fbRobot.bCNC_4_Reset := 		fbRobot.bCNC_4_Set;

fbRobot.bCNC_5_Reset := 		fbRobot.bCNC_5_Set AND
								stCNC5_Data^.DoorControl_DoorOpened AND
								(NOT stCNC5_Data^.DoorControl_Error) AND 
								stCNC5_Data^.ControlStatus_RobotModeActive
;

fbRobot(
	sName:= 'Fanuc - Satuzó', 
	bEn:= i_bLO2_CNC45, 
	timeBaseState:= T#40S, 
	bAck:= bAckP, 
	bOverride:= nOverride, 
	stEventArray:= arRobotEvents);
END_ACTION

END_PROGRAM

// ---- POUs/FBs/Fanuc/FB_Fanuc.TcPOU
FUNCTION_BLOCK FB_Fanuc
VAR_INPUT
	sName				:STRING;
	bEn					:BOOL;				(* Engedély jel *)
	eCommand			:E_Robot_Command;	(* Végrehajtandó parancsok *)	
	nViseNumber			:BYTE;				(* Satu sorszáma *)	
	nCncNumber			:BYTE;				(* CNC száma; 4 vagy 5 *)
	bVise_1_7_Reset		:BOOL;				(* Handshake *)
	bVise_8_14_Reset	:BOOL;				(* Handshake *)
	bCNC_4_Reset		:BOOL;				(* Handshake *)
	bCNC_5_Reset		:BOOL;				(* Handshake *)
	timeBaseState		:TIME:=T#20S;		(* Alaphelyzet felvételi idő*)
	bAck				:BOOL; 				(* Hibanyugta *)
	bOverride			:BYTE := 10;		(* PLC Override  10 - 100%*)
	stEventArray		:ARRAY [0..nMaxAlarmNr] OF TcEventEntry;	(* Event array definition *)
END_VAR
VAR_OUTPUT
	bReady				:BOOL;				(* Folyamat üzemkész *)
	bBusy				:BOOL;				(* Folyamat aktív *)
	bDone				:BOOL;				(* Folyamat kész *)
	bPendantMode		:BOOL;				(* Teach pendant mód aktív *)
	bVise_1_7_Set		:BOOL;				(* Handshake *)
	bVise_8_14_Set		:BOOL;				(* Handshake *)
	bCNC_4_Set			:BOOL;				(* Handshake *)
	bCNC_5_Set			:BOOL;				(* Handshake *)
	bError				:BOOL;				(* Hiba bit*)
	sError				:STRING(255);		(* Hiba string*)
END_VAR
VAR CONSTANT
	nMaxAlarmNr			:INT := 11;
END_VAR
VAR (* Robot IO *)
	RobotIn				:U_Fanuc_Input;
	RobotOut			:U_Fanuc_Output;
END_VAR
VAR (* State control *)
	tBaseState			:TON;
	tResetFault			:TON;
	tStopCycle			:TON;
	tStartCycle			:TON;
	
	nState				:UDINT;
	sState				:STRING;
	bIsInitalized		:BOOL;
	bRobotReady			:BOOL;
END_VAR
VAR (* Error handling*)
	bErrNotReady		:BOOL;
	bErrBaseTimeout		:BOOL;
	fbAlarmArray		:ARRAY [0..nMaxAlarmNr] OF FB_TcAlarm;
	arrAlarms			:ARRAY [0..nMaxAlarmNr] OF BOOL;
	i					:INT;
	
	//LastStates
	anLastStates				:ARRAY[0..500] OF UDINT;
    iLastStates					:INT;
END_VAR

(*Handshake**************************************************)
bVise_1_7_Set := RobotIn.Status.bVise_1_7_Set;
bVise_8_14_Set := RobotIn.Status.bVise_8_14_Set;
bCNC_4_Set := RobotIn.Status.bCNC_4_Set;
bCNC_5_Set := RobotIn.Status.bCNC_5_Set;
RobotOut.Control.bVise_1_7_Reset := bVise_1_7_Reset;
RobotOut.Control.bVise_8_14_Reset := bVise_8_14_Reset;
RobotOut.Control.bCNC_4_Reset := bCNC_4_Reset;
RobotOut.Control.bCNC_5_Reset := bCNC_5_Reset;

(*Időzítők***************************************************)
tBaseState(IN:= (nState > 0 AND nState < 10000), PT:= timeBaseState);
tResetFault(IN:= RobotOut.Control.bReset, PT:= T#100MS);
tStopCycle(IN:= RobotOut.Control.bCycleStop, PT:= T#100MS);
tStartCycle(IN:= RobotOut.Control.bStart, PT:= T#100MS);

(*Vész rendszer**************************************************)
bRobotReady :=  NOT RobotIn.Status.bControllerEmyStop AND
				NOT RobotIn.Status.bTeachPendantEmyStop AND
				NOT RobotIn.Status.bDeadman AND
				NOT RobotIn.Status.bFence AND
				NOT RobotIn.Status.bEmyStopExternal;
				
(*Hibakezelés************************************************)
IF nState >= 200 AND nState < 150000 AND (RobotIn.Status.bAlarm OR RobotIn.Status.bFault OR NOT bRobotReady) THEN
	bErrNotReady := TRUE;
END_IF

IF tBaseState.Q AND NOT bErrBaseTimeout THEN
	bErrBaseTimeout := TRUE;
END_IF

bError := (RobotIn.Status.bAlarm AND bEn) OR
			RobotIn.Status.bNoPneumatics OR
			RobotIn.Status.bNotCorrectPrg OR
			RobotIn.Status.bNotProductOnRobot OR
			RobotIn.Status.bProductOnRobot OR
			RobotIn.Status.bGripperOpenError OR
			RobotIn.Status.bGripperCloseError OR
			RobotIn.Status.bNotCorrectViseNumber OR
			bErrNotReady OR
			bErrBaseTimeout;

arrAlarms[0] := RobotIn.Status.bNoPneumatics;			
arrAlarms[1] := RobotIn.Status.bNotCorrectPrg;
arrAlarms[2] := RobotIn.Status.bNotProductOnRobot;
arrAlarms[3] := RobotIn.Status.bProductOnRobot;
arrAlarms[4] := RobotIn.Status.bGripperOpenError;
arrAlarms[5] := RobotIn.Status.bGripperCloseError;
arrAlarms[6] := RobotIn.Status.bNotCorrectViseNumber;
arrAlarms[7] := bErrNotReady;
arrAlarms[8] := bErrBaseTimeout;

IF nState > 140 AND nState < 150000 AND bError THEN
	nState := 200000;
END_IF
					
(*State history ************************************************)
IF(nState >= 100) AND (nState <= 20000) THEN
(*Steps before any state*)
	IF anLastStates[0] <> nState THEN
		FOR iLastStates:=500 TO 1 BY -1 DO
			anLastStates[iLastStates]:= anLastStates[iLastStates-1];
		END_FOR
		anLastStates[0]:= nState;
	END_IF
END_IF	

(*Pendant mód ************************************************)
bPendantMode := RobotIn.Status.bPendant;
IF bPendantMode THEN
	nState := 150000;
END_IF

(*Engedélyek *************************************************)
IF (NOT bEn AND NOT bPendantMode) THEN			// nincs ajtókör, és pendantról sem szeretnék használni
	nState := 0;
END_IF

// Enable signals
RobotOut.Control.bZoneEnable := bEn;
RobotOut.Control.bPlcOverride := bOverride;

(*Automata üzem *********************************************)
CASE nState OF
	(* Emergency circuit broken - Base state *)
	0:(* Operation stop - Emergency circuit check *)
		sState := CONCAT(UDINT_TO_STRING(nState) ,' - Vészkör vagy ajtókör bontva - Működtetések törlése');
		RobotOut.Control.bImmediateStop := FALSE;
		RobotOut.Control.bHold := FALSE;
		RobotOut.Control.bSafeSpeed := FALSE;
		RobotOut.Control.bCycleStop := FALSE;
		RobotOut.Control.bReset := FALSE;
		RobotOut.Control.bStart := FALSE;
		RobotOut.Control.bPNS1 := TRUE;
		RobotOut.Control.bPNS2 := FALSE;
		RobotOut.Control.bPNS3 := FALSE;
		RobotOut.Control.bPNS4 := FALSE;
		RobotOut.Control.bPNS5 := FALSE;
		RobotOut.Control.bPNS6 := FALSE;
		RobotOut.Control.bPNS7 := FALSE;
		RobotOut.Control.bPNS8 := FALSE;
		RobotOut.Control.bPnsStrobe := FALSE;
		RobotOut.Control.bEnable := FALSE;
		RobotOut.Control.bHome := FALSE;
		RobotOut.Control.bServiceEnd := FALSE;
		RobotOut.Control.nMode := 0;
		RobotOut.Control.nProgramNumber := 0;
		RobotOut.Control.bProdStart := FALSE;
		RobotOut.Control.bVise_1_7_Reset := FALSE;
		RobotOut.Control.bVise_8_14_Reset := FALSE;
		RobotOut.Control.bCNC_4_Reset := FALSE;
		RobotOut.Control.bCNC_5_Reset := FALSE;
		bErrNotReady := FALSE;
		bErrBaseTimeout := FALSE;
		bReady := FALSE;
		bBusy := FALSE;	
		IF bEn AND bRobotReady THEN
			bBusy := TRUE;
			nState := nState + 20;
		END_IF
		
	20:	
		sState := CONCAT(UDINT_TO_STRING(nState) ,' - Alaphelyzetfelvétel - Robot bekapcsolása');
		RobotOut.Control.bImmediateStop := TRUE;
		RobotOut.Control.bHold := TRUE;
		RobotOut.Control.bSafeSpeed := TRUE;
		RobotOut.Control.bEnable := TRUE;
		IF RobotIn.Status.bFault AND NOT RobotOut.Control.bReset THEN
			RobotOut.Control.bReset := TRUE;	// Ha hiba van -> Reset
		END_IF
		nState := nState + 20;

	40:
		sState := CONCAT(UDINT_TO_STRING(nState) ,' - Alaphelyzet felvétel - Robot hibatörlés');	
		IF tResetFault.Q THEN
			RobotOut.Control.bReset := FALSE;
		END_IF
		IF NOT RobotOut.Control.bReset AND NOT RobotIn.Status.bFault THEN
			nState := nState + 20;
		END_IF

	60:
		sState := CONCAT(UDINT_TO_STRING(nState) ,' - Alaphelyzet felvétel - Várakozás Robot hibatörlésre');	
		IF RobotIn.Status.bCommandEnable AND NOT RobotIn.Status.bFault THEN
			nState := nState + 20;
		END_IF
		
	80:
		sState := CONCAT(UDINT_TO_STRING(nState) ,' - Alaphelyzet felvétel - Robot Cycle Stop');
		RobotOut.Control.bCycleStop := TRUE;
		IF tStopCycle.Q THEN
			RobotOut.Control.bCycleStop := FALSE;
			nState := nState + 20;
		END_IF
	
	100:
		sState := CONCAT(UDINT_TO_STRING(nState) ,' - Alaphelyzet felvétel - Robot Cycle Start');
		RobotOut.Control.bStart := TRUE;
		IF tStartCycle.Q THEN
			RobotOut.Control.bStart := FALSE;
			nState := nState + 20;
		END_IF
		
	120: 
		sState := CONCAT(UDINT_TO_STRING(nState) ,' - Alaphelyzet felvétel - Várakozás Robot Cycle Start-ra');
		IF RobotIn.Status.bBusy AND RobotIn.Status.bProgramEnd THEN
			nState := nState + 20;
		END_IF
		
	140:
		sState := CONCAT(UDINT_TO_STRING(nState) ,' - Alaphelyzet felvétel - Alaphelyzet felvétel - Robot Busy');
		IF RobotIn.Status.bBusy THEN
			RobotOut.Control.bProdStart := TRUE;
			nState := nState + 20;
		END_IF
		
	160:
		sState := CONCAT(UDINT_TO_STRING(nState) ,' - Alaphelyzet felvétel - Robot alaphelyzetbe küldése');	
		RobotOut.Control.nProgramNumber := TO_BYTE(E_Robot_Programs.Home);
		IF RobotOut.Control.nProgramNumber = RobotIn.Status.nProgramNumber THEN
			RobotOut.Control.nProgramNumber := 0;
			nState := nState + 20;
		END_IF
		
	180:
		sState := CONCAT(UDINT_TO_STRING(nState) ,' - Alaphelyzet felvétel - Várakozás a robotprogram végére.');	
		IF RobotIn.Status.bProgramEnd AND NOT RobotIn.Status.bProgramRun THEN
			nState := nState + 20;
		END_IF
		
	200:
		nState := 10000;
		 
(* Alaphelyzet *********************************************************************)
	10000:
		sState := CONCAT(UDINT_TO_STRING(nState) ,' - Alaphelyzet - Várakozás parancsra');
		IF eCommand = E_Robot_Command.NoCommand THEN
			bReady := TRUE;
			bBusy := FALSE;
			bDone := FALSE;
		ELSE
			bReady := TRUE;
			bBusy := TRUE;
			bDone := FALSE;
			IF eCommand = E_Robot_Command.Home THEN			
				nState := 11000;	
			ELSIF eCommand = E_Robot_Command.Wait THEN	
				nState := 12000;
			ELSIF eCommand = E_Robot_Command.Service THEN	
				nState := 13000;
			ELSIF eCommand = E_Robot_Command.Pick_Up_Vise THEN	
				nState := 14000;
			ELSIF eCommand = E_Robot_Command.Put_Down_Vise THEN	
				nState := 15000;
			ELSIF eCommand = E_Robot_Command.Pick_Up_Cnc THEN	
				nState := 16000;
			ELSIF eCommand = E_Robot_Command.Put_Down_Cnc THEN	
				nState := 17000;
			ELSIF eCommand = E_Robot_Command.Move_To_Clean THEN	
				nState := 18000;
			END_IF
		END_IF

{region "Move to Home"} 
	(*-----=== Move to home program végrehajtása ===-----*)
	11000:	
		sState := CONCAT(UDINT_TO_STRING(nState) ,' - Robot alaphelyzetbe küldése');	
			 
		RobotOut.Control.nProgramNumber := TO_BYTE(E_Robot_Programs.Home);
			 
		IF RobotOut.Control.nProgramNumber = RobotIn.Status.nProgramNumber THEN
			RobotOut.Control.nProgramNumber := 0;
			nState := nState + 20;
		END_IF
		
	11020:
		sState := CONCAT(UDINT_TO_STRING(nState) ,' - Várakozás a robotprogram végére.');	
		IF RobotIn.Status.bProgramEnd AND NOT RobotIn.Status.bProgramRun THEN
			nState := nState + 20;
		END_IF
		
	11040:
		sState := CONCAT(UDINT_TO_STRING(nState) ,' - Várakozás mozgásparancs törlésére.');
		bReady := TRUE;
		bBusy := FALSE;
		bDone := TRUE;
		IF eCommand = E_Robot_Command.NoCommand THEN
			nState := 10000;
		END_IF
{enregion}
	 
{region "Move to Wait"}
	(*-----=== Move to wait program végrehajtása ===-----*)
	12000:	
		sState := CONCAT(UDINT_TO_STRING(nState) ,' - Robot várakozó pozícióba küldése');	
				  
		RobotOut.Control.nProgramNumber := TO_BYTE(E_Robot_Programs.Park);
				  
		IF RobotOut.Control.nProgramNumber = RobotIn.Status.nProgramNumber THEN
			RobotOut.Control.nProgramNumber := 0;
			nState := nState + 20;
		END_IF
		
	12020:
		sState := CONCAT(UDINT_TO_STRING(nState) ,' - Várakozás a robotprogram végére.');	
		IF RobotIn.Status.bProgramEnd AND NOT RobotIn.Status.bProgramRun THEN
			nState := nState + 20;
		END_IF
		
	12040:
		sState := CONCAT(UDINT_TO_STRING(nState) ,' - Várakozás mozgásparancs törlésére.');
		bReady := TRUE;
		bBusy := FALSE;
		bDone := TRUE;
		IF eCommand = E_Robot_Command.NoCommand THEN
			nState := 10000;
		END_IF
{enregion}
	 
{region "Move to Service"}
	(*-----=== Move to service program végrehajtása ===-----*)
	13000:	
		sState := CONCAT(UDINT_TO_STRING(nState) ,' - Robot szervíz pozícióba küldése');	
					   
		RobotOut.Control.nProgramNumber := TO_BYTE(E_Robot_Programs.Service);
					   
		IF RobotOut.Control.nProgramNumber = RobotIn.Status.nProgramNumber THEN
			RobotOut.Control.nProgramNumber := 0;
			nState := nState + 20;
		END_IF
		
	13020:
		sState := CONCAT(UDINT_TO_STRING(nState) ,' - Várakozás a robotprogram végére.');	
		IF RobotIn.Status.bProgramEnd AND NOT RobotIn.Status.bProgramRun THEN
			nState := nState + 20;
		END_IF
		
	13040:
		sState := CONCAT(UDINT_TO_STRING(nState) ,' - Várakozás mozgásparancs törlésére.');
		bReady := TRUE;
		bBusy := FALSE;
		bDone := TRUE;
		IF eCommand = E_Robot_Command.NoCommand THEN
			nState := 10000;
		END_IF
{enregion}
	 
{region "Pick up vise"}
	(*-----=== Pick up vise program végrehajtása ===-----*)
	14000:	
		sState := CONCAT(UDINT_TO_STRING(nState) ,' - Felvétel satuzóból');
							
		RobotOut.Control.nViseNumber := nViseNumber;
							
		IF nViseNumber <= 7 THEN
			RobotOut.Control.nProgramNumber := TO_BYTE(E_Robot_Programs.VisePickUp_1_7);
		ELSIF nViseNumber >= 8 THEN
			RobotOut.Control.nProgramNumber := TO_BYTE(E_Robot_Programs.VisePickUp_8_14);
		END_IF
							
		IF RobotOut.Control.nProgramNumber = RobotIn.Status.nProgramNumber THEN
			RobotOut.Control.nProgramNumber := 0;
			nState := nState + 20;
		END_IF
		
	14020:
		sState := CONCAT(UDINT_TO_STRING(nState) ,' - Várakozás a robotprogram végére.');	
		IF RobotIn.Status.bProgramEnd AND NOT RobotIn.Status.bProgramRun THEN
			nState := nState + 20;
		END_IF
		
	14040:
		sState := CONCAT(UDINT_TO_STRING(nState) ,' - Várakozás mozgásparancs törlésére.');
		bReady := TRUE;
		bBusy := FALSE;
		bDone := TRUE;
		IF eCommand = E_Robot_Command.NoCommand THEN
			nState := 10000;
		END_IF
{enregion}
	 
{region "Put down vise"}
	(*-----=== Put down vise program végrehajtása ===-----*)
	15000:	
		sState := CONCAT(UDINT_TO_STRING(nState) ,' - Lerakás satuzóba');
		RobotOut.Control.nViseNumber := nViseNumber;
		IF nViseNumber <= 7 THEN
			RobotOut.Control.nProgramNumber := TO_BYTE(E_Robot_Programs.VisePutDown_1_7);
		ELSIF nViseNumber >= 8 THEN
			RobotOut.Control.nProgramNumber := TO_BYTE(E_Robot_Programs.VisePutDown_8_14);
		END_IF
		IF RobotOut.Control.nProgramNumber = RobotIn.Status.nProgramNumber THEN
			RobotOut.Control.nProgramNumber := 0;
			nState := nState + 20;
		END_IF
		
	15020:
		sState := CONCAT(UDINT_TO_STRING(nState) ,' - Várakozás a robotprogram végére.');	
		IF RobotIn.Status.bProgramEnd AND NOT RobotIn.Status.bProgramRun THEN
			nState := nState + 20;
		END_IF
		
	15040:
		sState := CONCAT(UDINT_TO_STRING(nState) ,' - Várakozás mozgásparancs törlésére.');
		bReady := TRUE;
		bBusy := FALSE;
		bDone := TRUE;
		IF eCommand = E_Robot_Command.NoCommand THEN
			nState := 10000;
		END_IF
{enregion}
	 
{region "Pick up from CNC"}
	(*-----=== Pick up from CNC program végrehajtása ===-----*)
	16000:	
		sState := CONCAT(UDINT_TO_STRING(nState) ,' - Felvétel CNC-ből');
									  
		IF nCncNumber = 4 THEN
			RobotOut.Control.nProgramNumber := TO_BYTE(E_Robot_Programs.VisePickUpFromCnc_4);
		ELSE
			RobotOut.Control.nProgramNumber := TO_BYTE(E_Robot_Programs.VisePickUpFromCnc_5);
		END_IF
									  
		IF RobotOut.Control.nProgramNumber = RobotIn.Status.nProgramNumber THEN
			RobotOut.Control.nProgramNumber := 0;
			nState := nState + 20;
		END_IF
		
	16020:
		sState := CONCAT(UDINT_TO_STRING(nState) ,' - Várakozás a robotprogram végére.');	
		IF RobotIn.Status.bProgramEnd AND NOT RobotIn.Status.bProgramRun THEN
			nState := nState + 20;
		END_IF
		
	16040:
		sState := CONCAT(UDINT_TO_STRING(nState) ,' - Várakozás mozgásparancs törlésére.');
		bReady := TRUE;
		bBusy := FALSE;
		bDone := TRUE;
		IF eCommand = E_Robot_Command.NoCommand THEN
			nState := 10000;
		END_IF
{enregion}
	 
{region "Put down into CNC"}	
	(*-----=== Put down into CNC program végrehajtása ===-----*)
	17000:	
		sState := CONCAT(UDINT_TO_STRING(nState) ,' - Berakás CNC-be');
										   
		IF nCncNumber = 4 THEN
			RobotOut.Control.nProgramNumber := TO_BYTE(E_Robot_Programs.VisePutDownToCnc_4);
		ELSE
			RobotOut.Control.nProgramNumber := TO_BYTE(E_Robot_Programs.VisePutDownToCnc_5);
		END_IF
										   
		IF RobotOut.Control.nProgramNumber = RobotIn.Status.nProgramNumber THEN
			RobotOut.Control.nProgramNumber := 0;
			nState := nState + 20;
		END_IF
		
	17020:
		sState := CONCAT(UDINT_TO_STRING(nState) ,' - Várakozás a robotprogram végére.');	
		IF RobotIn.Status.bProgramEnd AND NOT RobotIn.Status.bProgramRun THEN
			nState := nState + 20;
		END_IF
		
	17040:
		sState := CONCAT(UDINT_TO_STRING(nState) ,' - Várakozás mozgásparancs törlésére.');
		bReady := TRUE;
		bBusy := FALSE;
		bDone := TRUE;
		IF eCommand = E_Robot_Command.NoCommand THEN
			nState := 10000;
		END_IF
{enregion}
	 
{region "Pendant mode"}
(* Pendant mód *********************************************************************)
	150000:	sState := CONCAT(UDINT_TO_STRING(nState) ,' - Pendant mód');
			IF NOT bPendantMode THEN
				RobotOut.Control.bImmediateStop := FALSE;
				RobotOut.Control.bHold := FALSE;
				RobotOut.Control.bZoneEnable := FALSE;
				RobotOut.Control.bEnable := FALSE;
				nState := 0;
			ELSE
				RobotOut.Control.bEnable := TRUE;
				RobotOut.Control.bHold := TRUE;
				RobotOut.Control.bZoneEnable := TRUE;
				RobotOut.Control.bImmediateStop := TRUE;
			END_IF
{endregion}
		
(* Hibakezelés *********************************************************************)
	200000:	sState := CONCAT(UDINT_TO_STRING(nState) ,CONCAT(' - Hiba, ebből az állapotból: ' ,sState));
			bReady := FALSE;
			bBusy := FALSE;	
			nState := nState + 20;

(* Hibakezelés *********************************************************************)
	200020:	
			IF bAck THEN			
				nState := nState + 20;
			END_IF
			
	200040: 
			RobotOut.Control.bImmediateStop := TRUE;
			RobotOut.Control.bReset := TRUE;
			RobotOut.Control.bNotCorrectPrg_Reset := TRUE;
			RobotOut.Control.bNotProductOnRobot_Reset := TRUE;
			RobotOut.Control.bProductOnRobot_Reset := TRUE;
			RobotOut.Control.bGripperOpenError_Reset := TRUE;
			RobotOut.Control.bGripperCloseError_Reset := TRUE;
			RobotOut.Control.bNotCorrectViseNumber_Reset := TRUE;
			nState := nState + 20;
			
	200060:
			IF 	NOT RobotIn.Status.bNoPneumatics AND
				NOT RobotIn.Status.bNotCorrectPrg AND
				NOT RobotIn.Status.bNotProductOnRobot AND
				NOT RobotIn.Status.bProductOnRobot AND
				NOT RobotIn.Status.bGripperOpenError AND
				NOT RobotIn.Status.bGripperCloseError AND
				NOT RobotIn.Status.bNotCorrectViseNumber
			THEN
				nState := nState + 20;
			END_IF	
			
	200080:
			RobotOut.Control.bReset := FALSE;
			RobotOut.Control.bNotCorrectPrg_Reset := FALSE;
			RobotOut.Control.bNotProductOnRobot_Reset := FALSE;
			RobotOut.Control.bProductOnRobot_Reset := FALSE;
			RobotOut.Control.bGripperOpenError_Reset := FALSE;
			RobotOut.Control.bGripperCloseError_Reset := FALSE;
			RobotOut.Control.bNotCorrectViseNumber_Reset := FALSE;
			bErrNotReady := FALSE;
			bErrBaseTimeout := FALSE;
			nState := 0;
ELSE
	sState := CONCAT(UDINT_TO_STRING(nState) ,' - Nem használt állapot');
END_CASE	


(*Hiba string*)
IF bError THEN
	sError := sName;
	FOR i:=0 TO nMaxAlarmNr DO
		IF arrAlarms[i] THEN
			IF (fbAlarmArray[i].eConfirmationState <> 2 AND fbAlarmArray[i].nTimeCleared <> 0 AND fbAlarmArray[i].nTimeConfirmed <> 0) OR //Ha már volt alarm, akkor van bennük érték
				(fbAlarmArray[i].eConfirmationState = 1 AND fbAlarmArray[i].nTimeCleared = 0 AND fbAlarmArray[i].nTimeConfirmed = 0)	//Első futás esetén
			THEN
				fbAlarmArray[i].Raise(0);
			END_IF
		END_IF
	END_FOR 
ELSE
	sError := '';
END_IF

(*Hiba kezelés Tc3_EventLogger*)
IF NOT bIsInitalized THEN
	bIsInitalized := TRUE;
	FOR i:=0 TO nMaxAlarmNr DO
		fbAlarmArray[i].CreateEx(stEventArray[i], TRUE, 0);
	END_FOR
END_IF

(*Hiba törlés (nyugtázott és megszűnt)*)
FOR i:=0 TO nMaxAlarmNr DO
	IF fbAlarmArray[i].eConfirmationState = 3 AND NOT bError THEN
		fbAlarmArray[i].Clear(0, FALSE);
	END_IF
END_FOR

END_FUNCTION_BLOCK

// ---- POUs/Temp/Robot.TcPOU
PROGRAM Robot
VAR
	tResetFault					:TON;
	tStopCycle					:TON;
	tStartCycle					:TON;
END_VAR

(*Bemetek olvasása*******************************************)
stFanucIn := uFanucIn.stFanucIn;
stDigiForceIn := uDigiForceIn.stDigiforce_In;
(*Időzítők***************************************************)
tResetFault(IN:= stFanucOut.stCtrl.bReset, PT:= T#100MS);
tStopCycle(IN:= stFanucOut.stCtrl.bCycleStop, PT:= T#100MS);
tStartCycle(IN:= stFanucOut.stCtrl.bStart, PT:= T#100MS);
(*Triggerek**************************************************)

(*Vész rendszer**********************************************)
bRobotReady := 	NOT stFanucIn.stEmergency.bEMGOP AND
				NOT	stFanucIn.stEmergency.bEMGTP AND
				NOT	stFanucIn.stEmergency.bDEADMAN AND
				NOT	stFanucIn.stEmergency.bFENCE AND
				NOT	stFanucIn.stEmergency.bEMGEX;
				
IF	NOT i_bLOp2 AND
	stRobot.nState > 0 THEN
			stRobot.nState := 0;
END_IF
(*Hibakezelés************************************************)
bRobotAlarm := stRobot.nState > 140 AND	(stFanucIn.stAlarm.bAlarm1 OR
										stFanucIn.stAlarm.bAlarm2 OR
										stFanucIn.stAlarm.bAlarm3 OR
										stFanucIn.stAlarm.bAlarm4 OR
										stFanucIn.stAlarm.bAlarm5 OR
										stFanucIn.stAlarm.bAlarm6);

IF stRobot.nState > 60 AND stRobot.nState < 150000 THEN
	stRobot.nStateLast := stRobot.nState;
	IF	stFanucIn.stCtrl.bFault OR bRobotAlarm OR NOT bRobotReady THEN
			stRobot.nState := 200000;
	END_IF
END_IF
										
(*Engedélyek *************************************************)
IF stRobot.nState <= 10000
	OR stRobot.nState = 150000
	OR stRobot.nState >= 200000
THEN
	stRobot.bManualModeEnable := TRUE;
ELSE
	stRobot.bManualModeEnable := FALSE;
END_IF

IF stRobot.nState = 0
	OR stRobot.nState = 10000
	OR stRobot.nState = 150000
	OR stRobot.nState >= 200000
THEN
	stRobot.bDoorOpenEnable := TRUE;
ELSE
	stRobot.bDoorOpenEnable := FALSE;
END_IF

(*Kézi üzem *************************************************)
IF bManualModeVise and stRobot.nState < 150000 THEN
	stRobot.nState := 150000;
END_IF

(*Automata üzem *********************************************)
CASE stRobot.nState OF
	0:		IF i_bLOp2 AND stProcessReq.bEco THEN			
				stRobot.sState := CONCAT(UDINT_TO_STRING(stRobot.nState) ,' - Robot "ECO" mód aktív - Működtetések törlése');
			ELSE
				stRobot.sState := CONCAT(UDINT_TO_STRING(stRobot.nState) ,' - Vészkör vagy ajtókör bontva - Működtetések törlése');				
			END_IF
			stFanucOut.stCtrl.bImStop := FALSE; 
			stFanucOut.stCtrl.bHold := FALSE; 
			stFanucOut.stCtrl.bSafetyfSpeed := FALSE; 
			stFanucOut.stCtrl.bCycleStop := FALSE; 
			stFanucOut.stCtrl.bReset := FALSE; 
			stFanucOut.stCtrl.bStart := FALSE; 
			stFanucOut.stCtrl.bEnable := FALSE; 
			stFanucOut.stCtrl.bPsr1 := FALSE; 
			stFanucOut.stCtrl.bPsr2 := FALSE; 
			stFanucOut.stCtrl.bPsr3 := FALSE; 
			stFanucOut.stCtrl.bPsr4 := FALSE; 
			stFanucOut.stCtrl.bPsrStrobe := FALSE;
			stFanucOut.stCtrl.bMoveEnable := FALSE; 
			stFanucOut.stCtrl.bServiceEnd := FALSE;
			stFanucOut.stProg.nType := 0;
			stFanucOut.stProg.nMode := 0;
			stFanucOut.stProg.nProgNr := 0;
			stProcessReq.bExecute := FALSE;
			stProcessReq.nProgIdx := 0;
			stRobot.bError := 0;
			IF i_bLOp2 AND bRobotReady AND NOT stProcessReq.bEco THEN
				IF bStepEnable THEN
					stRobot.nState := stRobot.nState + 20;
				END_IF
			END_IF

	20:		stRobot.sState := CONCAT(UDINT_TO_STRING(stRobot.nState) ,' - Alaphelyzet felvétel - Robot bekapcsolása');
			stFanucOut.stCtrl.bImStop := TRUE; 
			stFanucOut.stCtrl.bHold := TRUE; 
			stFanucOut.stCtrl.bSafetyfSpeed := TRUE; 
			stFanucOut.stCtrl.bEnable := TRUE;
			IF stFanucIn.stCtrl.bFault AND NOT stFanucOut.stCtrl.bReset THEN
				stFanucOut.stCtrl.bReset := TRUE;									// Ha hiba van -> Reset
			END_IF
			IF bStepEnable THEN
				stRobot.nState := stRobot.nState + 20;
			END_IF

	40:		stRobot.sState := CONCAT(UDINT_TO_STRING(stRobot.nState) ,' - Alaphelyzet felvétel - Robot hibatörlés');
			IF tResetFault.Q THEN
				stFanucOut.stCtrl.bReset := FALSE;									// Timer-re kell törölni! Hanshake nincs.
			END_IF
			IF NOT stFanucIn.stCtrl.bFault AND NOT stFanucOut.stCtrl.bReset THEN
				IF bStepEnable THEN
					stRobot.nState := stRobot.nState + 20;							// Ha se hiba se reset akkor mehet tovább.
				END_IF
			END_IF
			
	60:		stRobot.sState := CONCAT(UDINT_TO_STRING(stRobot.nState) ,' - Alaphelyzet felvétel - Várakozás Robot hibatörlésre');
			IF stFanucIn.stCtrl.bCmdEnable AND NOT stFanucIn.stCtrl.bFault THEN
				IF bStepEnable THEN
					stRobot.nState := stRobot.nState + 20;
				END_IF
			END_IF

	80:		stRobot.sState := CONCAT(UDINT_TO_STRING(stRobot.nState) ,' - Alaphelyzet felvétel - Robot Cycle Stop');
			stFanucOut.stCtrl.bCycleStop := TRUE;
			IF tStopCycle.Q THEN
				stFanucOut.stCtrl.bCycleStop := FALSE;
				IF bStepEnable THEN
					stRobot.nState := stRobot.nState + 20;
				END_IF
			END_IF
	
	100:	stRobot.sState := CONCAT(UDINT_TO_STRING(stRobot.nState) ,' - Alaphelyzet felvétel - Robot Cycle Start');
			stFanucOut.stCtrl.bStart := TRUE;
			IF tStartCycle.Q THEN
				stFanucOut.stCtrl.bStart := FALSE;
				IF bStepEnable THEN
					stRobot.nState := stRobot.nState + 20;
				END_IF
			END_IF

			
	120:	stRobot.sState := CONCAT(UDINT_TO_STRING(stRobot.nState) ,' - Alaphelyzet felvétel - Várakozás Robot Cycle Start-ra');
			IF stFanucIn.stCtrl.bBusy AND stFanucIn.stCtrl.bProgEnd THEN
				IF bStepEnable THEN
					stRobot.nState := stRobot.nState + 20;
				END_IF
			END_IF
			
	140:	stRobot.sState := CONCAT(UDINT_TO_STRING(stRobot.nState) ,' - Alaphelyzet felvétel - Robot Busy');
			IF stFanucIn.stCtrl.bBusy THEN
				stFanucOut.stCtrl.bMoveEnable := TRUE;								// Robot mozgásengedély
				IF bStepEnable THEN
					stRobot.nState := stRobot.nState + 20;
				END_IF
			END_IF
			
	160:	stRobot.sState := CONCAT(UDINT_TO_STRING(stRobot.nState) ,' - Alaphelyzet felvétel - Robot alaphelyzetbe küldése');
			stFanucOut.stProg.nType := 1;
			stFanucOut.stProg.nMode := 1;
			stFanucOut.stProg.nProgNr := 1;
			IF stFanucOut.stProg.nProgNr = stFanucIn.stProg.nActProg THEN
				stFanucOut.stProg.nProgNr := 0;
				IF bStepEnable THEN
					stRobot.nState := stRobot.nState + 20;
				END_IF
			END_IF

	180:	stRobot.sState := CONCAT(UDINT_TO_STRING(stRobot.nState) ,' - Alaphelyzet felvétel - Várakozás a robotprogram végére.');
			IF	stFanucIn.stProg.nActPoint = 1 AND							// A robot a kiválsztott pontban van
				NOT stFanucIn.stCtrl.bProgRun AND							// A program nem fut
				stFanucIn.stCtrl.bProgEnd THEN								// A program végzett
					IF bStepEnable THEN
						stRobot.nState := stRobot.nState + 20;
					END_IF
			END_IF

	200:
			stRobot.nState := 10000;

	(* Alaphelyzet *********************************************************************)
	10000:	stRobot.sState := CONCAT(UDINT_TO_STRING(stRobot.nState) ,' - Alaphelyzet, parancsra vár');
			IF		stProcessReq.bEco THEN									// Eco mode vagy ajtónyitás
						IF bStepEnable THEN
							stRobot.nState := 20000;
						END_IF
			ELSIF	stProcessReq.bExecute THEN								// Program végrehajtás
						IF stProcessReq.nProgIdx > 0 THEN
							IF bStepEnable THEN
								stRobot.nState := 11000;
							END_IF
						ELSE
							stProcessReq.bExecute := FALSE;
						END_IF
			END_IF

(*-----=== Execute robot program ===-----*)			
	11000:	stRobot.sState := CONCAT(UDINT_TO_STRING(stRobot.nState) ,arrFanucReq[stProcessReq.nProgIdx].sName);
			stFanucOut.stProg.nType := word_to_byte(stP0.stFixtureData.nPcbType);
			stFanucOut.stProg.nMode := 1;
			stFanucOut.stProg.nProgNr := arrFanucReq[stProcessReq.nProgIdx].nProgNr;
			IF (stFanucOut.stProg.nProgNr = stFanucIn.stProg.nActProg) AND											//	A programot tükrözze vissza a robot és	(* Z.Zs. 2022.05.10. *)
			   (stFanucIn.stCtrl.bProgRun AND NOT stFanucIn.stCtrl.bProgEnd) THEN									//	indúljon el a mozgás is, mert a profinet és a PLC elég gyors ahoz, hogy a robotba még ne indúljon el a mozgás!!!!! 
				stProcessReq.nProgIdx := 0;
				IF stProcessReq.nProgIdx2 <> 0 THEN
					stFanucOut.stProg.nProgNr := arrFanucReq[stProcessReq.nProgIdx2].nProgNr;
					IF bStepEnable THEN
						stRobot.nState := stRobot.nState + 20;
					END_IF
				ELSE
					stFanucOut.stProg.nProgNr := 0;
					IF bStepEnable THEN
						stRobot.nState := stRobot.nState + 40;
					END_IF
				END_IF		
			END_IF
			
	11020:	stRobot.sState := CONCAT(UDINT_TO_STRING(stRobot.nState) ,arrFanucReq[stProcessReq.nProgIdx2].sName);
			IF stFanucOut.stProg.nProgNr = stFanucIn.stProg.nActProg THEN
				stProcessReq.nProgIdx2 := 0;
				stFanucOut.stProg.nProgNr := 0;
				IF bStepEnable THEN
					stRobot.nState := stRobot.nState + 20;
				END_IF
			END_IF

	11040:	stRobot.sState := CONCAT(UDINT_TO_STRING(stRobot.nState) ,' - Várakozás a robotprogram végére.');
			IF	NOT stFanucIn.stCtrl.bProgRun AND stFanucIn.stCtrl.bProgEnd THEN
				IF bStepEnable THEN
					stRobot.nState := stRobot.nState + 20;
				END_IF
			END_IF
	
	11060:	
			stRobot.nState := 50000;

(*-----=== ECO mode ===-----*)
	20000:	stRobot.sState := CONCAT(UDINT_TO_STRING(stRobot.nState) ,' - Robot Cycle Stop');
			stFanucOut.stCtrl.bCycleStop := TRUE;
			stFanucOut.stCtrl.bMoveEnable := FALSE;
			IF tStopCycle.Q THEN
				stFanucOut.stCtrl.bCycleStop := FALSE;
				IF bStepEnable THEN
					stRobot.nState := stRobot.nState + 20;
				END_IF
			END_IF

	20020:	stRobot.sState := CONCAT(UDINT_TO_STRING(stRobot.nState) ,' - Robot kikapcsolása');
			stFanucOut.stCtrl.bImStop := FALSE; 
			stFanucOut.stCtrl.bHold := FALSE; 
			stFanucOut.stCtrl.bSafetyfSpeed := FALSE; 
			stFanucOut.stCtrl.bEnable := FALSE;
			IF bStepEnable THEN
				stRobot.nState := 0;
			END_IF			
		
	50000:
			stProcessReq.nProgIdx := 0;
			stProcessReq.bExecute := FALSE;
			stRobot.nState := 10000;
	

	(* Kézi üzem *********************************************************************)
	150000:	stRobot.sState := CONCAT(UDINT_TO_STRING(stRobot.nState) ,' - Kézi üzem');
			IF NOT bManualModeVise THEN
				stRobot.nState := 0;
			ELSIF	stProcessReq.bExecute AND NOT bRobotAlarm AND bRobotReady THEN							// Program végrehajtás
						IF stProcessReq.nProgIdx > 0 THEN
							IF bStepEnable THEN
								stRobot.nState := 151000;
							END_IF
						ELSE
							stProcessReq.bExecute := FALSE;
						END_IF
			ELSIF bRobotAlarm THEN
					stRobot.nState := 152000;
			END_IF

(*-----=== Execute robot program ===-----*)			
	151000:	stRobot.sState := CONCAT(UDINT_TO_STRING(stRobot.nState) ,arrFanucReq[stProcessReq.nProgIdx].sName);
			stFanucOut.stProg.nType := WORD_TO_BYTE(stP0.stFixtureData.nPcbType);
			stFanucOut.stProg.nMode := 1;
			stFanucOut.stProg.nProgNr := arrFanucReq[stProcessReq.nProgIdx].nProgNr;
			IF stFanucOut.stProg.nProgNr = stFanucIn.stProg.nActProg THEN
				stFanucOut.stProg.nProgNr := 0;
				IF bStepEnable THEN
					stRobot.nState := stRobot.nState + 20;
				END_IF
			END_IF

	151020:	stRobot.sState := CONCAT(UDINT_TO_STRING(stRobot.nState) ,' - Várakozás a robotprogram végére.');
			IF	(NOT stFanucIn.stCtrl.bProgRun AND stFanucIn.stCtrl.bProgEnd) OR bRobotAlarm OR NOT bRobotReady THEN
				IF bStepEnable THEN
					stRobot.nState := stRobot.nState + 20;
				END_IF
			END_IF
	
	151040:
			stProcessReq.bExecute := FALSE;
			stRobot.nState := 150000;

(*-----=== Robot alarm törlése ===-----*)
	152000:
			stFanucOut.stAlarm.bAlarm1 := stFanucIn.stAlarm.bAlarm1;
			stFanucOut.stAlarm.bAlarm2 := stFanucIn.stAlarm.bAlarm2;
			stFanucOut.stAlarm.bAlarm3 := stFanucIn.stAlarm.bAlarm3;
			stFanucOut.stAlarm.bAlarm4 := stFanucIn.stAlarm.bAlarm4;
			stFanucOut.stAlarm.bAlarm5 := stFanucIn.stAlarm.bAlarm5;
			stFanucOut.stAlarm.bAlarm6 := stFanucIn.stAlarm.bAlarm6;
			IF NOT bRobotAlarm THEN
				stProcessReq.bExecute := FALSE;
				stRobot.nState := 150000;
			END_IF
	

	(* Hibakezelés *********************************************************************)
	200000:	stRobot.sState := CONCAT(UDINT_TO_STRING(stRobot.nState) ,CONCAT(' - Hiba, ebből az állapotból: ' ,stRobot.sState));
			stRobot.bError := TRUE;
			stRobot.nState := stRobot.nState + 20;

	(* Hibakezelés *********************************************************************)
	200020:	IF bAckP THEN
				stRobot.nState := stRobot.nState + 20;
			END_IF
			

	200040:	stFanucOut.stAlarm.bAlarm1 := stFanucIn.stAlarm.bAlarm1;
			stFanucOut.stAlarm.bAlarm2 := stFanucIn.stAlarm.bAlarm2;
			stFanucOut.stAlarm.bAlarm3 := stFanucIn.stAlarm.bAlarm3;
			stFanucOut.stAlarm.bAlarm4 := stFanucIn.stAlarm.bAlarm4;
			stFanucOut.stAlarm.bAlarm5 := stFanucIn.stAlarm.bAlarm5;
			stFanucOut.stAlarm.bAlarm6 := stFanucIn.stAlarm.bAlarm6;
			IF NOT bRobotAlarm THEN
				stRobot.nState := stRobot.nState + 20;
			END_IF
				
	200060:
				CASE stRobot.nStateLast OF
					(* Alaphelyzet felvétel folyamán *)
					0..9999:	stRobot.nState := 0;
				ELSE 			stRobot.nState := 0;
				END_CASE
				stRobot.bError := FALSE;
ELSE
	stRobot.sState := CONCAT(UDINT_TO_STRING(stRobot.nState) ,' - Nem használt állapot');
END_CASE


(*Robot handshake********************************************)
HandShake();
(*Kimetek írása**********************************************)
uFanucOut.stFanucOut := stFanucOut;
uDigiForceOut.stDigiforce_Out := stDigiForceOut;

ACTION HandShake:
stFanucOut.stHandShake.bFeederEnable := stFanucIn.stHandShake.bFeederReq;
stFanucOut.stHandShake.bPositioner1Enable := stFanucIn.stHandShake.bPositioner1Req;
stFanucOut.stHandShake.bPositioner2Enable := stFanucIn.stHandShake.bPositioner2Req;
stFanucOut.stHandShake.bFixtureAreaEnable := stFanucIn.stHandShake.bFixtureAreaReq;
stFanucOut.stHandShake.bPositioner1Open := stFanucIn.stHandShake.bPositioner1OpenReq AND fbP0Positioner1.bBasePosStab AND fbP0Positioner2.bBasePosStab;
stFanucOut.stHandShake.bPositioner2Open := stFanucIn.stHandShake.bPositioner2OpenReq AND fbP0Positioner3.bBasePosStab AND fbP0Positioner4.bBasePosStab;
END_ACTION

END_PROGRAM

// ---- POUs/Robot7AxisStation/Robot7AxisProgram.TcPOU
PROGRAM Robot7AxisProgram
VAR	(* Control *)
	nState						: UDINT;
	nStatePrevious				: UDINT;
	sState						: STRING(500);
	bError						: BOOL;
	fbCycleTime					: TON;
	nCycleTime					: REAL;
END_VAR
VAR //LastStates
	anLastStates				:ARRAY[0..500] OF UDINT;
    iLastStates					:INT;
END_VAR
VAR (* Robot *)
	fbRobot						: FB_Fanuc_CNC;
	arRobotEvents				: ARRAY [0..15] OF TcEventEntry;
END_VAR
VAR (* Test variables *)
	nOverride					: BYTE := 30;
	bTestEnable					: BOOL;
	nTestIndex					: BYTE;
	nTestCncIndex				: BYTE;
	bCamTest					: BOOL;
	rtCamReset					: R_TRIG;
	nProgNr						: UINT;
	nDimX						: LREAL;
	nDimY						: LREAL;
	nDimZ						: LREAL;
	nPosX						: LREAL;
	nPosY						: LREAL;
	nWeight						: UINT;
	nTorque						: REAL;
	nErrorId					: UDINT;
	ePath						: E_CNC_Robot_Path;
END_VAR
VAR	(*Communication with CNC-s*)
	bStartCNC1					:	BOOL;
	bStartCNC2					:	BOOL;
	bStartCNC3					:	BOOL;
	nPlaceBackFromThisCNC		:	BYTE;
END_VAR
VAR // MySQL
	
END_VAR

MySQL();
Camera();
rtCamReset(CLK:= bCamTest);

IF rtCamReset.Q THEN
		fb3DCam.ResetCam();
END_IF
IF bCamTest THEN
	IF fb3DCam.CamCheck(nProgNr, nDimX, nDimY, nDimZ, nErrorId) THEN
		bCamTest := FALSE;
	END_IF
END_IF

(*Error handling*)
IF nState > 0 AND nState < 150000 THEN
	nStatePrevious := nState;
END_IF

(*Maintance*)
IF bManualMode THEN
	nState := 150000;
END_IF

(*Emergency*)
IF NOT i_bLO1_Main THEN
	nState := 0;
END_IF

(*Last states*)
IF(nState >= 1000) AND (nState < 150000) THEN
(*Steps before any state*)
	IF anLastStates[0] <> nState THEN
		FOR iLastStates:=500 TO 1 BY -1 DO
			anLastStates[iLastStates]:= anLastStates[iLastStates-1];
		END_FOR
		anLastStates[0]:= nState;
	END_IF
END_IF	

IF fbRobot.bError
THEN
	bError  :=  TRUE;
END_IF


(*Yet, constantly write the offset to the used value, because it is the only needed offset now AT 2023.11.17.*)
nPosX := 62.5;
nPosY := (nDimX+4)/2+1;


CASE nState OF
{region "Alaphelyzet felvétel"}
	(****************************************************************************************)
	(******************************* Alaphelyzetfelvétel ************************************)
	(****************************************************************************************)	
	0:		(*-----=== Kimenetek törlése ===-----*)
		sState := CONCAT(UDINT_TO_STRING(nState) ,' - A biztonsági kör nem aktív');
			 
		fbRobot.eCommand := E_CNC_Robot_Command.NoCommand;
		bStartCNC1 := FALSE;
		bStartCNC2 := FALSE;
		bStartCNC3 := FALSE;	
		nPlaceBackFromThisCNC := 0;
			 
		IF i_bLO1_Main AND NOT bManualMode AND NOT fbRobot.bPendantMode THEN
			nState := nState + 20;
		END_IF

	20: 
		sState := CONCAT(UDINT_TO_STRING(nState) ,' - Robot alaphelyzetfelvétel');
		fbRobot.eCommand := E_CNC_Robot_Command.Home;
		IF NOT fbRobot.bBusy AND fbRobot.bReady THEN
			fbRobot.eCommand := E_CNC_Robot_Command.NoCommand;
			nState := nState + 20;
		END_IF

	40:
		nState := 10000;
{endregion}
	 

	10000:
		nState := 10500;
		
	10500:	
		sState := CONCAT(UDINT_TO_STRING(nState) ,' - Paletta kivétel-beküldés ellenőrzés');
		
		//Mi van ha megszakad a folyamat valami maitt?  Akkor is jó ha itt kezd? 
		
		IF stDutData_Cnc1.bDone AND (CNC_1.stCNC_Data^.DoorControl_DoorOpened AND (NOT CNC_1.bCNCHandshakeTimeout)) AND ((fbLift_1A.nTagID = stDutData_Cnc1.nPaletteId)OR(fbLift_1B.nTagID = stDutData_Cnc1.nPaletteId))THEN	//CNC Done, and CNC Door Opened
			
			
			IF fbLift_1A.nTagID = stDutData_Cnc1.nPaletteId THEN	//Decide that what lift should be used
				ePath := E_CNC_Robot_Path.CNC1_to_Lift1A;
				nPlaceBackFromThisCNC := 1;
				nState := 11000;
			ELSIF fbLift_1B.nTagID = stDutData_Cnc1.nPaletteId THEN
				ePath := E_CNC_Robot_Path.CNC1_to_Lift1B;
				nPlaceBackFromThisCNC := 2;
				nState := 11000;
			ELSE
				sState := CONCAT(UDINT_TO_STRING(nState) ,' - Ismeretlen cél lift paletta lerakáskor CNC 1 - Paletta Lift 1 A-B között');
			END_IF
			
		ELSIF stDutData_Cnc2.bDone AND (CNC_2.stCNC_Data^.DoorControl_DoorOpened AND (NOT CNC_2.bCNCHandshakeTimeout)) AND ((fbLift_2A.nTagID = stDutData_Cnc2.nPaletteId)OR(fbLift_2B.nTagID = stDutData_Cnc2.nPaletteId))THEN //CNC Done, and CNC Door Opened
			
			
			IF fbLift_2A.nTagID = stDutData_Cnc2.nPaletteId THEN	//Decide that what lift should be used
				ePath := E_CNC_Robot_Path.CNC2_to_Lift2A;
				nPlaceBackFromThisCNC := 3;
				nState := 11000;
			ELSIF fbLift_2B.nTagID = stDutData_Cnc2.nPaletteId THEN
				ePath := E_CNC_Robot_Path.CNC2_to_Lift2B;
				nPlaceBackFromThisCNC := 4;
				nState := 11000;
			ELSE
				sState := CONCAT(UDINT_TO_STRING(nState) ,' - Ismeretlen cél lift paletta lerakáskor CNC 2 - Paletta Lift 2 A-B között');
			END_IF
		
		ELSIF stDutData_Cnc3.bDone AND (CNC_3.stCNC_Data^.DoorControl_DoorOpened AND (NOT CNC_3.bCNCHandshakeTimeout)) AND ((fbLift_3A.nTagID = stDutData_Cnc3.nPaletteId)OR(fbLift_3B.nTagID = stDutData_Cnc3.nPaletteId))THEN //CNC Done, and CNC Door Opened
				
			nPlaceBackFromThisCNC := 3;
			IF fbLift_3A.nTagID = stDutData_Cnc3.nPaletteId THEN	//Decide that what lift should be used
				ePath := E_CNC_Robot_Path.CNC3_to_Lift3A;
				nPlaceBackFromThisCNC := 5;
				nState := 11000;
			ELSIF fbLift_3B.nTagID = stDutData_Cnc3.nPaletteId THEN
				ePath := E_CNC_Robot_Path.CNC3_to_Lift3B;
				nPlaceBackFromThisCNC := 6;
				nState := 11000;
			ELSE
				sState := CONCAT(UDINT_TO_STRING(nState) ,' - Ismeretlen cél lift paletta lerakáskor CNC 3 - Paletta Lift 3 A-B között');
			END_IF	
			
		
		ELSIF  (NOT CNC_1.bCNCRunning) AND (CNC_1.stCNC_Data^.DoorControl_DoorOpened AND (NOT CNC_1.bCNCHandshakeTimeout)) AND (GVL_Palette.arrPalette[fbLift_1A.nTagID].nState = 3) THEN //Pallet is at the stopper, CNC not running, CNC door is opened
		 		stDutData_Cnc1 := GVL_Palette.arrPalette[fbLift_1A.nTagID];
				ePath := E_CNC_Robot_Path.Lift1A_to_CNC1;
				bStartCNC1 := TRUE;
				nState := 11000;
		ELSIF  (NOT CNC_1.bCNCRunning) AND (CNC_1.stCNC_Data^.DoorControl_DoorOpened AND (NOT CNC_1.bCNCHandshakeTimeout)) AND (GVL_Palette.arrPalette[fbLift_1B.nTagID].nState = 3 ) THEN //Pallet is at the stopper, CNC not running, CNC door is opened
		 		stDutData_Cnc1 := GVL_Palette.arrPalette[fbLift_1B.nTagID];
				ePath := E_CNC_Robot_Path.Lift1B_to_CNC1;
				bStartCNC1 := TRUE;
				nState := 11000;
			
			
		ELSIF  (NOT CNC_2.bCNCRunning) AND (CNC_2.stCNC_Data^.DoorControl_DoorOpened AND (NOT CNC_2.bCNCHandshakeTimeout)) AND (GVL_Palette.arrPalette[fbLift_2A.nTagID].nState = 3)THEN //Pallet is at the stopper, CNC not running, CNC door is opened
		 		stDutData_Cnc2 := GVL_Palette.arrPalette[fbLift_2A.nTagID];
				ePath := E_CNC_Robot_Path.Lift2A_to_CNC2;
				bStartCNC2 := TRUE;
				nState := 11000;
		ELSIF  (NOT CNC_2.bCNCRunning) AND (CNC_2.stCNC_Data^.DoorControl_DoorOpened AND (NOT CNC_2.bCNCHandshakeTimeout)) AND (GVL_Palette.arrPalette[fbLift_2B.nTagID].nState = 3)THEN //Pallet is at the stopper, CNC not running, CNC door is opened
		 		stDutData_Cnc2 := GVL_Palette.arrPalette[fbLift_2B.nTagID];
				ePath := E_CNC_Robot_Path.Lift2B_to_CNC2;
				bStartCNC2 := TRUE;
				nState := 11000;
			
			
		ELSIF  (NOT CNC_3.bCNCRunning) AND (CNC_3.stCNC_Data^.DoorControl_DoorOpened AND (NOT CNC_3.bCNCHandshakeTimeout)) AND (GVL_Palette.arrPalette[fbLift_3A.nTagID].nState = 3) THEN //Pallet is at the stopper, CNC not running, CNC door is opened
		 		stDutData_Cnc3 := GVL_Palette.arrPalette[fbLift_3A.nTagID];
				ePath := E_CNC_Robot_Path.Lift3A_to_CNC3;
				bStartCNC3 := TRUE;
				nState := 11000;
		ELSIF  (NOT CNC_3.bCNCRunning) AND (CNC_3.stCNC_Data^.DoorControl_DoorOpened AND (NOT CNC_3.bCNCHandshakeTimeout)) AND (GVL_Palette.arrPalette[fbLift_3B.nTagID].nState = 3) THEN //Pallet is at the stopper, CNC not running, CNC door is opened
		 		stDutData_Cnc3 := GVL_Palette.arrPalette[fbLift_3B.nTagID];
				ePath := E_CNC_Robot_Path.Lift3B_to_CNC3;
				bStartCNC3 := TRUE;
				nState := 11000;
		END_IF
		

		
{region "Alaphelyzet"}
	(****************************************************************************************)
	(*********************************** Alaphelyzet ****************************************)
	(****************************************************************************************)	
	11000:		(* -----=== Várakozás parancsra ===----- *)
		sState := CONCAT(UDINT_TO_STRING(nState) ,' - Alaphelyzet');
		CASE ePath OF
			E_CNC_Robot_Path.Lift1A_to_CNC1:
												nProgNr := 1;
												fbRobot.nCncNumber := 1;
												fbRobot.eLifterNumber := E_Lifter.Lifter_1A;
												nDimX := stDutData_Cnc1.nDimX;
												nDimY := stDutData_Cnc1.nDimY;
												nDimZ := stDutData_Cnc1.nDimZ;
												nPosX := stDutData_Cnc1.nPosX;
												nPosY := stDutData_Cnc1.nPosY;
												nWeight := stDutData_Cnc1.nWeight;
												nTorque := stDutData_Cnc1.nTorque;
//												stDutData_Cnc1.nDutId := 1;
												nState := 20000;
			E_CNC_Robot_Path.CNC1_to_Lift1A:
												fbRobot.nCncNumber := 1;
												fbRobot.eLifterNumber := E_Lifter.Lifter_1A;
												fbRobot.nOffset_X := nPosX;
												fbRobot.nOffset_Y := nPosY;
												fbRobot.nWeight := stDutData_Cnc1.nWeight;	
												nState := 30000;

			E_CNC_Robot_Path.Lift1B_to_CNC1:
												nProgNr := 2;
												fbRobot.nCncNumber := 1;
												fbRobot.eLifterNumber := E_Lifter.Lifter_1B;
												nDimX := stDutData_Cnc1.nDimX;
												nDimY := stDutData_Cnc1.nDimY;
												nDimZ := stDutData_Cnc1.nDimZ;
												nPosX := stDutData_Cnc1.nPosX;
												nPosY := stDutData_Cnc1.nPosY;
												nWeight := stDutData_Cnc1.nWeight;
												nTorque := stDutData_Cnc1.nTorque;
//												stDutData_Cnc1.nDutId := 1;
												nState := 20000;

			E_CNC_Robot_Path.CNC1_to_Lift1B:
												fbRobot.nCncNumber := 1;
												fbRobot.eLifterNumber := E_Lifter.Lifter_1B;
												fbRobot.nOffset_X := nPosX;
												fbRobot.nOffset_Y := nPosY;
												fbRobot.nWeight := stDutData_Cnc1.nWeight;
												nState := 30000;
													 
														  
															   
																	
																		 
													 
			E_CNC_Robot_Path.Lift2A_to_CNC2:
												nProgNr := 3;
												fbRobot.nCncNumber := 2;
												fbRobot.eLifterNumber := E_Lifter.Lifter_2A;
												nDimX := stDutData_Cnc2.nDimX;
												nDimY := stDutData_Cnc2.nDimY;
												nDimZ := stDutData_Cnc2.nDimZ;
												nPosX := stDutData_Cnc2.nPosX;
												nPosY := stDutData_Cnc2.nPosY;
												nWeight := stDutData_Cnc2.nWeight;
												nTorque := stDutData_Cnc2.nTorque;
//												stDutData_Cnc2.nDutId := 1;
												nState := 20000;
			E_CNC_Robot_Path.CNC2_to_Lift2A:
												fbRobot.nCncNumber := 2;
												fbRobot.eLifterNumber := E_Lifter.Lifter_2A;
												fbRobot.nOffset_X := nPosX;
												fbRobot.nOffset_Y := nPosY;
												fbRobot.nWeight := stDutData_Cnc2.nWeight;	
												nState := 30000;

			E_CNC_Robot_Path.Lift2B_to_CNC2:
												nProgNr := 4;
												fbRobot.nCncNumber := 2;
												fbRobot.eLifterNumber := E_Lifter.Lifter_2B;
												nDimX := stDutData_Cnc2.nDimX;
												nDimY := stDutData_Cnc2.nDimY;
												nDimZ := stDutData_Cnc2.nDimZ;
												nPosX := stDutData_Cnc2.nPosX;
												nPosY := stDutData_Cnc2.nPosY;
												nWeight := stDutData_Cnc2.nWeight;
												nTorque := stDutData_Cnc2.nTorque;
//												stDutData_Cnc2.nDutId := 1;
												nState := 20000;

			E_CNC_Robot_Path.CNC2_to_Lift2B:
												fbRobot.nCncNumber := 2;
												fbRobot.eLifterNumber := E_Lifter.Lifter_2B;
												fbRobot.nOffset_X := nPosX;
												fbRobot.nOffset_Y := nPosY;
												fbRobot.nWeight := stDutData_Cnc2.nWeight;
												nState := 30000;
													 
														  
															   
																	
																		 
																			  
																				   
			E_CNC_Robot_Path.Lift3A_to_CNC3:
												nProgNr := 5;
												fbRobot.nCncNumber := 3;
												fbRobot.eLifterNumber := E_Lifter.Lifter_3A;
												nDimX := stDutData_Cnc3.nDimX;
												nDimY := stDutData_Cnc3.nDimY;
												nDimZ := stDutData_Cnc3.nDimZ;
												nPosX := stDutData_Cnc3.nPosX;
												nPosY := stDutData_Cnc3.nPosY;
												nWeight := stDutData_Cnc3.nWeight;
												nTorque := stDutData_Cnc3.nTorque;
//												stDutData_Cnc3.nDutId := 1;
												nState := 20000;
			E_CNC_Robot_Path.CNC3_to_Lift3A:
												fbRobot.nCncNumber := 3;
												fbRobot.eLifterNumber := E_Lifter.Lifter_3A;
												fbRobot.nOffset_X := nPosX;
												fbRobot.nOffset_Y := nPosY;
												fbRobot.nWeight := stDutData_Cnc3.nWeight;	
												nState := 30000;

			E_CNC_Robot_Path.Lift3B_to_CNC3:
												nProgNr := 6;
												fbRobot.nCncNumber := 3;
												fbRobot.eLifterNumber := E_Lifter.Lifter_3B;
												nDimX := stDutData_Cnc3.nDimX;
												nDimY := stDutData_Cnc3.nDimY;
												nDimZ := stDutData_Cnc3.nDimZ;
												nPosX := stDutData_Cnc3.nPosX;
												nPosY := stDutData_Cnc3.nPosY;
												nWeight := stDutData_Cnc3.nWeight;
												nTorque := stDutData_Cnc3.nTorque;
//												stDutData_Cnc3.nDutId := 1;
												nState := 20000;

			E_CNC_Robot_Path.CNC3_to_Lift3B:
												fbRobot.nCncNumber := 3;
												fbRobot.eLifterNumber := E_Lifter.Lifter_3B;
												fbRobot.nOffset_X := nPosX;
												fbRobot.nOffset_Y := nPosY;
												fbRobot.nWeight := stDutData_Cnc3.nWeight;
												nState := 30000;
		END_CASE
{endregion}

{region "bepakolás a CNC-be"}
	(****************************************************************************************)
	(********************************** Kiemelő -> CNC **************************************)
	(****************************************************************************************)
	20000:		(*-----=== Szkennelési pozícióba ===-----*)
		sState := CONCAT(UDINT_TO_STRING(nState) ,' - Robot kamara pozícióba');
		
		bStartCNC1 := FALSE;
		bStartCNC2 := FALSE;
		bStartCNC3 := FALSE;	 
		
		fbRobot.nOffset_X := 0;
		fbRobot.nOffset_Y := 0;
		fbRobot.nOffset_Z := 0;
		fbRobot.nOffset_W := 0;
		fbRobot.nOffset_P := 0;
		fbRobot.nOffset_R := 0;
		fbRobot.eCommand := E_CNC_Robot_Command.Camera_Lifter;
		IF fbRobot.bBusy THEN
			ePath := E_CNC_Robot_Path.NoPath;
			nState := nState + 20;
		END_IF
		
	20020:		(*-----=== Várakozás Robotmozgásra ===-----*)
		sState := CONCAT(UDINT_TO_STRING(nState) ,' - Várakozáas robot mozgásra');
		IF NOT fbRobot.bBusy THEN
			fbRobot.eCommand := E_CNC_Robot_Command.NoCommand;
			fb3DCam.ResetCam();
			nState := nState + 20;
		END_IF

	20040:		(*-----=== 3D kamera triggerelése ===-----*)
		sState := CONCAT(UDINT_TO_STRING(nState) ,' - 3D kamera triggerelése');
		IF fb3DCam.CamCheck(nProgNr, nDimX, nDimY, nDimZ, nErrorId) THEN
			IF fb3DCam.p_Pass THEN
				nState := nState + 20;
			ELSE
				nState := 200000;
			END_IF
		END_IF

	20060:		(*-----=== Darabfelvétel ===-----*)
		sState := CONCAT(UDINT_TO_STRING(nState) ,' - Robot felvételi pozícióba');
		fbRobot.nOffset_X := fb3DCam.p_PosX;
		fbRobot.nOffset_Y := fb3DCam.p_PosY;
		fbRobot.nOffset_Z := fb3DCam.p_PosZ;
		fbRobot.nOffset_W := fb3DCam.p_PosW;
		fbRobot.nOffset_P := fb3DCam.p_PosP;
		fbRobot.nOffset_R := fb3DCam.p_PosR;
		fbRobot.eCommand := E_CNC_Robot_Command.Pick_Up_Lifter;
		IF fbRobot.bBusy THEN
			nState := nState + 20;
		END_IF
		
	20080:		(*-----=== Várakozás Robotmozgásra ===-----*)
		sState := CONCAT(UDINT_TO_STRING(nState) ,' - Várakozáas robot mozgásra');
		IF NOT fbRobot.bBusy THEN
			fbRobot.eCommand := E_CNC_Robot_Command.NoCommand;
			fb3DCam.ResetCam();
			nState := nState + 20;
		END_IF

	20100:		(*-----=== Darab lerakása ===-----*)
		sState := CONCAT(UDINT_TO_STRING(nState) ,' - Darab lerakása CNC1-be');
		nPosX := 62.5;
		nPosY := (nDimX+4)/2+1;
		fbRobot.nOffset_X := nPosX;
		fbRobot.nOffset_Y := nPosY;
		fbRobot.nOffset_Z := 0;
		fbRobot.nOffset_W := 0;
		fbRobot.nOffset_P := 0;
		fbRobot.nOffset_R := 0;
		fbRobot.eCommand := E_CNC_Robot_Command.Put_Down_CNC;
		IF fbRobot.bBusy THEN
			nState := nState + 20;
		END_IF
		
	20120:		(*-----=== Várakozás Robotmozgásra ===-----*)
		sState := CONCAT(UDINT_TO_STRING(nState) ,' - Várakozáas robot mozgásra');
			   
		IF NOT fbRobot.bBusy THEN
			fbRobot.eCommand := E_CNC_Robot_Command.NoCommand;
			fb3DCam.ResetCam();
			nState := nState + 20;
		END_IF

	20140:		(*-----=== Robot QuickHome pozícióba ===-----*)
		sState := CONCAT(UDINT_TO_STRING(nState) ,' - Robot HOME pozícióba');
		fbRobot.nOffset_X := 0;
		fbRobot.nOffset_Y := 0;
		fbRobot.nOffset_Z := 0;
		fbRobot.nOffset_W := 0;
		fbRobot.nOffset_P := 0;
		fbRobot.nOffset_R := 0;
		fbRobot.eCommand := E_CNC_Robot_Command.QuickHome;
		IF fbRobot.bBusy THEN
			nState := nState + 20;
		END_IF
		
	20160:		(*-----=== Várakozás Robotmozgásra ===-----*)
		sState := CONCAT(UDINT_TO_STRING(nState) ,' - Várakozáas robot mozgásra');
		IF NOT fbRobot.bBusy THEN
			fbRobot.eCommand := E_CNC_Robot_Command.NoCommand;
			fb3DCam.ResetCam();
			nState := nState + 20;
		END_IF

	20180:
		nState := 10000;
{endregion}

{region "kipakolás a CNC-ből"}
	(****************************************************************************************)
	(********************************** CNC -> Kiemelő **************************************)
	(****************************************************************************************)
	30000:		(*-----=== CNC pozícióba ===-----*)
		sState := CONCAT(UDINT_TO_STRING(nState) ,' - Robot CNC pozícióba');
		fbRobot.eCommand := E_CNC_Robot_Command.Pick_Up_CNC;
		IF fbRobot.bBusy THEN
			ePath := E_CNC_Robot_Path.NoPath;
			nState := nState + 20;
		END_IF

	30020:		(*-----=== Várakozás Robotmozgásra ===-----*)
		sState := CONCAT(UDINT_TO_STRING(nState) ,' - Várakozáas robot mozgásra');
		IF NOT fbRobot.bBusy THEN
			fbRobot.eCommand := E_CNC_Robot_Command.NoCommand;
			fb3DCam.ResetCam();
			nState := nState + 20;
		END_IF

	30040:		(*-----=== Lift pozícióba ===-----*)
		sState := CONCAT(UDINT_TO_STRING(nState) ,' - Robot Lift pozícióba');
		fbRobot.eCommand := E_CNC_Robot_Command.Put_Down_Lifter;
		IF fbRobot.bBusy THEN
			nState := nState + 20;
		END_IF

	30060:		(*-----=== Várakozás Robotmozgásra ===-----*)
		sState := CONCAT(UDINT_TO_STRING(nState) ,' - Várakozáas robot mozgásra');
			 
		IF NOT fbRobot.bBusy THEN
					   
			//Liftek visszaküldése alaphelyzetbe			  
			IF nPlaceBackFromThisCNC = 1 THEN
				stDutData_Cnc1.nState.3 := TRUE;
				GVL_Palette.arrPalette[stDutData_Cnc1.nPaletteId].nState.3 := TRUE;
				GVL_Palette.arrPalette[stDutData_Cnc1.nPaletteId].nTarget := 7;
			ELSIF nPlaceBackFromThisCNC = 2 THEN
				stDutData_Cnc1.nState.3 := TRUE;	
				GVL_Palette.arrPalette[stDutData_Cnc1.nPaletteId].nState.3 := TRUE;
				GVL_Palette.arrPalette[stDutData_Cnc1.nPaletteId].nTarget := 7;
					 
			ELSIF nPlaceBackFromThisCNC = 3 THEN
				stDutData_Cnc2.nState.3 := TRUE; 
				GVL_Palette.arrPalette[stDutData_Cnc2.nPaletteId].nState.3 := TRUE;
				GVL_Palette.arrPalette[stDutData_Cnc1.nPaletteId].nTarget := 7;
			ELSIF nPlaceBackFromThisCNC = 4 THEN
				stDutData_Cnc2.nState.3 := TRUE; 
				GVL_Palette.arrPalette[stDutData_Cnc2.nPaletteId].nState.3 := TRUE;
				GVL_Palette.arrPalette[stDutData_Cnc1.nPaletteId].nTarget := 7;
					 
			ELSIF nPlaceBackFromThisCNC = 5 THEN
				stDutData_Cnc3.nState.3 := TRUE; 
				GVL_Palette.arrPalette[stDutData_Cnc3.nPaletteId].nState.3 := TRUE;
				GVL_Palette.arrPalette[stDutData_Cnc1.nPaletteId].nTarget := 7;
			ELSIF nPlaceBackFromThisCNC = 6 THEN
				stDutData_Cnc3.nState.3 := TRUE; 
				GVL_Palette.arrPalette[stDutData_Cnc3.nPaletteId].nState.3 := TRUE;
				GVL_Palette.arrPalette[stDutData_Cnc1.nPaletteId].nTarget := 7;
			END_IF			  
							  		   
		
			fbRobot.eCommand := E_CNC_Robot_Command.NoCommand;
			fb3DCam.ResetCam();
			nState := nState + 20;
		END_IF

	30080:		(*-----=== Robot QuickHome pozícióba ===-----*)
		sState := CONCAT(UDINT_TO_STRING(nState) ,' - Robot HOME pozícióba');
		fbRobot.nOffset_X := 0;
		fbRobot.nOffset_Y := 0;
		fbRobot.nOffset_Z := 0;
		fbRobot.nOffset_W := 0;
		fbRobot.nOffset_P := 0;
		fbRobot.nOffset_R := 0;
		fbRobot.eCommand := E_CNC_Robot_Command.QuickHome;
		IF fbRobot.bBusy THEN
			nState := nState + 20;
		END_IF
		
	30100:		(*-----=== Várakozás Robotmozgásra ===-----*)
		sState := CONCAT(UDINT_TO_STRING(nState) ,' - Várakozáas robot mozgásra');
		IF NOT fbRobot.bBusy THEN
			fbRobot.eCommand := E_CNC_Robot_Command.NoCommand;
			fb3DCam.ResetCam();
			nState := nState + 20;
		END_IF

	30120:
		nState := 10000;


	
	150000: (* Maintenance *)
		sState := CONCAT(UDINT_TO_STRING(nState) ,' - Maintenance');
		IF NOT bManualMode THEN
			nState := 0;
		END_IF
		
	200000:(* Error handling *)
		sState := CONCAT(UDINT_TO_STRING(nState) ,CONCAT(' - Error, from this state: ' , sState));
		nState := 200020;

	200020:(* Error handling *)
		IF bAckP THEN
			CASE nStatePrevious OF
				0..9999: nState := 0;
//				10000..25000: nState := 10000;
//				30000..31000: nState := 30000;
			ELSE nState := 0;
			END_CASE
		END_IF	
		
	ELSE //Not a real step, for test purposes
		sState := CONCAT(UDINT_TO_STRING(nState) ,' - Not a real step, for test purposes');
END_CASE

(*Timers***************************************************)
fbCycleTime(IN:= nState > 10000 AND nState <= 95000, PT:= T#1D, Q=> , ET=> );
IF nState > 10000 AND nState <= 95000 THEN
	nCycleTime := TIME_TO_REAL(fbCycleTime.ET)/1000;
END_IF

Robot();

ACTION Camera:
fb3DCam();
END_ACTION

ACTION MySQL:
;
END_ACTION

ACTION Robot:
arRobotEvents[0] := TC_EVENTS.MyEvents.RobotNoPneumaticsErr;
arRobotEvents[1] := TC_EVENTS.MyEvents.RobotNotCorrectPrgErr;
arRobotEvents[2] := TC_EVENTS.MyEvents.RobotNotProdOnRobotErr;
arRobotEvents[3] := TC_EVENTS.MyEvents.RobotProdOnRobotErr;
arRobotEvents[4] := TC_EVENTS.MyEvents.RobotGripperOpenErr;
arRobotEvents[5] := TC_EVENTS.MyEvents.RobotGripperCloseErr;
arRobotEvents[6] := TC_EVENTS.MyEvents.RobotNotCorrectViseNumberErr;
arRobotEvents[7] := TC_EVENTS.MyEvents.RobotNotReadyErr;
arRobotEvents[8] := TC_EVENTS.MyEvents.RobotBasePosErr;

(*-----=== Gripper jelek kezelése ===-----*)
fbGripperPos1(
	nCalOffset:= 34.9, 
	nReqDistance:= nDimY, 
	bPendantMode:= fbRobot.bPendantMode, 
	bValid=> , 
	nDistance=> , 
	bGripperInPos=> );

fbGripperPos2(
	nCalOffset:= 35, 
	nReqDistance:= nDimY, 
	bPendantMode:= fbRobot.bPendantMode, 
	bValid=> , 
	nDistance=> , 
	bGripperInPos=> );



(*-----=== Hand shake jelek kezelése ===-----*)
fbRobot.bCNC_1_Reset := 			fbRobot.bCNC_1_Set AND				// 05.1	Robot CNC-1-be menne
									i_bRobotDoorOpened_CNC1 AND
									CNC_1.nState = 11100 OR CNC_1.nState = 12000;

fbRobot.bCNC_1_ViseClose_Reset := 	fbRobot.bCNC_1_ViseClose_Set AND	// 05.2	Robot CNC-1 satu zárásra vár
									CNC_1.nState = 11300;

fbRobot.bCNC_1_ViseOpen_Reset := 	fbRobot.bCNC_1_ViseOpen_Set AND		// 05.3	Robot CNC-1 satu nyitásra vár
									CNC_1.nState = 12000;

fbRobot.bCNC_2_Reset := 			fbRobot.bCNC_2_Set AND				// 05.4	Robot CNC-2-be menne
									i_bRobotDoorOpened_CNC2;

fbRobot.bCNC_2_ViseClose_Reset := 	fbRobot.bCNC_2_ViseClose_Set;		// 05.5	Robot CNC-2 satu zárásra vár

fbRobot.bCNC_2_ViseOpen_Reset := 	fbRobot.bCNC_2_ViseOpen_Set;		// 05.6	Robot CNC-2 satu nyitásra vár

fbRobot.bCNC_3_Reset := 			fbRobot.bCNC_3_Set AND				// 05.7	Robot CNC-3-be menne
									i_bRobotDoorOpened_CNC3;

fbRobot.bCNC_3_ViseClose_Reset := 	fbRobot.bCNC_3_ViseClose_Set;		// 05.8	Robot CNC-3 satu zárásra vár
	
fbRobot.bCNC_3_ViseOpen_Reset := 	fbRobot.bCNC_3_ViseOpen_Set;		// 06.1	Robot CNC-3 satu nyitásra vár

fbRobot.bPalette_1_Reset := 		fbRobot.bPalette_1_Set;				// 06.2	Robot Kiemelő 1-hez menne

fbRobot.bPalette_2_Reset := 		fbRobot.bPalette_2_Set;				// 06.3	Robot Kiemelő 2-höz menne

fbRobot.bPalette_3_Reset := 		fbRobot.bPalette_3_Set;				// 06.4	Robot Kiemelő 3-hoz menne

fbRobot.bGripperClosed_Reset := 	fbRobot.bGripperClosed_Set AND		// 06.5	Robot megfogó zárás SET
									(fbGripperPos1.bGripperInPos OR
									fbGripperPos2.bGripperInPos);


fbRobot(
	sName:= 'Fanuc - 7 axis', 
	bEn:= i_bLO2_Main, 
	timeBaseState:= T#40S, 
	bAck:= bAckP, 
	bOverride:= nOverride, 
	stEventArray:= arRobotEvents);
END_ACTION

END_PROGRAM

// ---- POUs/FBs/FanucCNC/FB_Fanuc_CNC.TcPOU
FUNCTION_BLOCK FB_Fanuc_CNC
VAR_INPUT
	sName					:STRING;
	bEn						:BOOL;				(* Engedély jel *)
	eCommand				:E_CNC_Robot_Command;(* Végrehajtandó parancsok *)	
	nCncNumber				:BYTE;				(* CNC gép sorszáma (1-3) *)
	eLifterNumber			:E_Lifter;			(* Kiemelő stípusa *)
	nWeight					:UINT;				(* Offszet érték *)
	nOffset_ID				:UINT;				(* Offszet érték *)
	nOffset_X				:REAL;				(* X tengelyű offszet érték *)
	nOffset_Y				:REAL;				(* Y tengelyű offszet érték *)
	nOffset_Z				:REAL;				(* Z tengelyű offszet érték *)
	nOffset_W				:REAL;				(* W tengelyű offszet érték *)
	nOffset_P				:REAL;				(* P tengelyű offszet érték *)
	nOffset_R				:REAL;				(* R tengelyű offszet érték *)
	bCNC_1_Reset			:BOOL;				(* Handshake *)
	bCNC_1_ViseClose_Reset	:BOOL;				(* Handshake *)
	bCNC_1_ViseOpen_Reset	:BOOL;				(* Handshake *)
	bCNC_2_Reset			:BOOL;				(* Handshake *)
	bCNC_2_ViseClose_Reset	:BOOL;				(* Handshake *)
	bCNC_2_ViseOpen_Reset	:BOOL;				(* Handshake *)
	bCNC_3_Reset			:BOOL;				(* Handshake *)
	bCNC_3_ViseClose_Reset	:BOOL;				(* Handshake *)
	bCNC_3_ViseOpen_Reset	:BOOL;				(* Handshake *)
	bPalette_1_Reset		:BOOL;				(* Handshake *)
	bPalette_2_Reset		:BOOL;				(* Handshake *)
	bPalette_3_Reset		:BOOL;				(* Handshake *)
	bGripperClosed_Reset	:BOOL;				(* Handshake *)
	timeBaseState			:TIME:=T#20S;		(* Alaphelyzet felvételi idő*)
	bAck					:BOOL; 				(* Hibanyugta *)
	bOverride				:BYTE := 10;		(* PLC Override  10 - 100%*)
	stEventArray			:ARRAY [0..nMaxAlarmNr] OF TcEventEntry;	(* Event array definition *)
END_VAR
VAR_OUTPUT
	bReady					:BOOL;				(* Folyamat üzemkész *)
	bBusy					:BOOL;				(* Folyamat aktív *)
	bDone					:BOOL;				(* Folyamat kész *)
	bPendantMode			:BOOL;				(* Teach pendant mód aktív *)
	bCNC_1_Set				:BOOL;				(* Handshake *)
	bCNC_1_ViseClose_Set	:BOOL;				(* Handshake *)
	bCNC_1_ViseOpen_Set		:BOOL;				(* Handshake *)
	bCNC_2_Set				:BOOL;				(* Handshake *)
	bCNC_2_ViseClose_Set	:BOOL;				(* Handshake *)
	bCNC_2_ViseOpen_Set		:BOOL;				(* Handshake *)
	bCNC_3_Set				:BOOL;				(* Handshake *)
	bCNC_3_ViseClose_Set	:BOOL;				(* Handshake *)
	bCNC_3_ViseOpen_Set		:BOOL;				(* Handshake *)
	bPalette_1_Set			:BOOL;				(* Handshake *)
	bPalette_2_Set			:BOOL;				(* Handshake *)
	bPalette_3_Set			:BOOL;				(* Handshake *)
	bGripperClosed_Set		:BOOL;				(* Handshake *)
	bError					:BOOL;				(* Hiba bit*)
	sError					:STRING(255);		(* Hiba string*)
	bZoneCnc1				:BOOL;				(* Robot bent a területen Zone 1*)
	bZoneCnc2				:BOOL;				(* Robot bent a területen Zone 2*)
	bZoneCnc3				:BOOL;				(* Robot bent a területen Zone 3*)
	bZoneLift1				:BOOL;				(* Robot bent a területen Zone 4*)
	bZoneLift2				:BOOL;				(* Robot bent a területen Zone 5*)
	bZoneLift3				:BOOL;				(* Robot bent a területen Zone 6*)
	bZoneGudel				:BOOL;				(* Robot bent a területen Zone 7*)
	bZoneMaster				:BOOL;				(* Robot bent a területen Zone 8*)
	nOffset_ID_Echo			:UINT;				(* Offszet érték *)
	nOffset_X_Echo			:REAL;				(* X tengelyű offszet érték *)
	nOffset_Y_Echo			:REAL;				(* Y tengelyű offszet érték *)
	nOffset_Z_Echo			:REAL;				(* Z tengelyű offszet érték *)
	nOffset_W_Echo			:REAL;				(* W tengelyű offszet érték *)
	nOffset_P_Echo			:REAL;				(* P tengelyű offszet érték *)
	nOffset_R_Echo			:REAL;				(* R tengelyű offszet érték *)
END_VAR
VAR CONSTANT
	nMaxAlarmNr			:INT := 15;
	nDecimalPlaces		:USINT := 3;
END_VAR
VAR (* Robot IO *)
	RobotIn				:U_CNC_Fanuc_Input;
	RobotOut			:U_CNC_Fanuc_Output;
END_VAR
VAR (* State control *)
	tBaseState			:TON;
	tResetFault			:TON;
	tStopCycle			:TON;
	tStartCycle			:TON;
	
	nState				:UDINT;
	sState				:STRING;
	bIsInitalized		:BOOL;
	bRobotReady			:BOOL;
END_VAR
VAR (* Error handling*)
	bErrNotReady		:BOOL;
	bErrBaseTimeout		:BOOL;
	fbAlarmArray		:ARRAY [0..nMaxAlarmNr] OF FB_TcAlarm;
	arrAlarms			:ARRAY [0..nMaxAlarmNr] OF BOOL;
	i					:INT;
	
	//LastStates
	anLastStates				:ARRAY[0..500] OF UDINT;
    iLastStates					:INT;
END_VAR
VAR
// TEST !!!!!!!!!!!!!!!!!!!!!!
	bTestConvert		: BOOL;
END_VAR

(*Test*) //TÖRÖLNI HA MÁR HOMÁR!!!!!!!!!!!!!!!!!!!!!!!!!!!!!!!!!!!!!!!!!!!!!!!!!!!!!!!!!!!!!!!!!!!!!!!!!!!!!!!!!!!!!!!
IF bTestConvert THEN
		REAL_TO_WHOLE_AND_FRACTION(nReal := nOffset_X,
									nWhole => RobotOut.Control.nOffset_X_Whole,
									nFraction => RobotOut.Control.nOffset_X_Fractional);
		REAL_TO_WHOLE_AND_FRACTION(nReal := nOffset_Y,
									nWhole => RobotOut.Control.nOffset_Y_Whole,
									nFraction => RobotOut.Control.nOffset_Y_Fractional);
		REAL_TO_WHOLE_AND_FRACTION(nReal := nOffset_Z,
									nWhole => RobotOut.Control.nOffset_Z_Whole,
									nFraction => RobotOut.Control.nOffset_Z_Fractional);
		REAL_TO_WHOLE_AND_FRACTION(nReal := nOffset_W,
									nWhole => RobotOut.Control.nOffset_W_Whole,
									nFraction => RobotOut.Control.nOffset_W_Fractional);
		REAL_TO_WHOLE_AND_FRACTION(nReal := nOffset_P,
									nWhole => RobotOut.Control.nOffset_P_Whole,
									nFraction => RobotOut.Control.nOffset_P_Fractional);
		REAL_TO_WHOLE_AND_FRACTION(nReal := nOffset_R,
									nWhole => RobotOut.Control.nOffset_R_Whole,
									nFraction => RobotOut.Control.nOffset_R_Fractional);
		bTestConvert := FALSE;
END_IF
(*Offset Echo************************************************)
nOffset_ID_Echo := RobotIn.Status.nOffset_ID;
WHOLE_AND_FRACTION_TO_REAL(nWhole:= RobotIn.Status.nOffset_X_Whole, nFraction:=RobotIn.Status.nOffset_X_Fractional, nReal=> nOffset_X_Echo);
WHOLE_AND_FRACTION_TO_REAL(nWhole:= RobotIn.Status.nOffset_Y_Whole, nFraction:=RobotIn.Status.nOffset_Y_Fractional, nReal=> nOffset_Y_Echo);
WHOLE_AND_FRACTION_TO_REAL(nWhole:= RobotIn.Status.nOffset_Z_Whole, nFraction:=RobotIn.Status.nOffset_Z_Fractional, nReal=> nOffset_Z_Echo);
WHOLE_AND_FRACTION_TO_REAL(nWhole:= RobotIn.Status.nOffset_W_Whole, nFraction:=RobotIn.Status.nOffset_W_Fractional, nReal=> nOffset_W_Echo);
WHOLE_AND_FRACTION_TO_REAL(nWhole:= RobotIn.Status.nOffset_P_Whole, nFraction:=RobotIn.Status.nOffset_P_Fractional, nReal=> nOffset_P_Echo);
WHOLE_AND_FRACTION_TO_REAL(nWhole:= RobotIn.Status.nOffset_R_Whole, nFraction:=RobotIn.Status.nOffset_R_Fractional, nReal=> nOffset_R_Echo);

(*Handshake**************************************************)
bCNC_1_Set := RobotIn.Status.bCNC_1_Set;
bCNC_1_ViseClose_Set := RobotIn.Status.bCNC_1_ViseClose_Set;
bCNC_1_ViseOpen_Set := RobotIn.Status.bCNC_1_ViseOpen_Set;
bCNC_2_Set := RobotIn.Status.bCNC_2_Set;
bCNC_2_ViseClose_Set := RobotIn.Status.bCNC_2_ViseClose_Set;
bCNC_2_ViseOpen_Set := 	RobotIn.Status.bCNC_2_ViseOpen_Set;
bCNC_3_Set := RobotIn.Status.bCNC_3_Set;
bCNC_3_ViseClose_Set := RobotIn.Status.bCNC_3_ViseClose_Set;
bCNC_3_ViseOpen_Set := RobotIn.Status.bCNC_3_ViseOpen_Set;
bPalette_1_Set := RobotIn.Status.bPalette_1_Set;
bPalette_2_Set := RobotIn.Status.bPalette_2_Set;
bPalette_3_Set := RobotIn.Status.bPalette_3_Set;
bGripperClosed_Set := RobotIn.Status.bGripperClosed_Set;
RobotOut.Control.bCNC_1_Reset := bCNC_1_Reset;
RobotOut.Control.bCNC_1_ViseClose_Reset := bCNC_1_ViseClose_Reset;
RobotOut.Control.bCNC_1_ViseOpen_Reset := bCNC_1_ViseOpen_Reset;
RobotOut.Control.bCNC_2_Reset := bCNC_2_Reset;
RobotOut.Control.bCNC_2_ViseClose_Reset := bCNC_2_ViseClose_Reset;
RobotOut.Control.bCNC_2_ViseOpen_Reset := 	bCNC_2_ViseOpen_Reset;
RobotOut.Control.bCNC_3_Reset := bCNC_3_Reset;
RobotOut.Control.bCNC_3_ViseClose_Reset := bCNC_3_ViseClose_Reset;
RobotOut.Control.bCNC_3_ViseOpen_Reset := bCNC_3_ViseOpen_Reset;
RobotOut.Control.bPalette_1_Reset := bPalette_1_Reset;
RobotOut.Control.bPalette_2_Reset := bPalette_2_Reset;
RobotOut.Control.bPalette_3_Reset := bPalette_3_Reset;
RobotOut.Control.bGripperClosed_Reset := bGripperClosed_Reset;
RobotOut.Control.nWeight := nWeight;

(*Zónák******************************************************)
bZoneCnc1 :=  RobotIn.Status.bZone_1_CNC_1;
bZoneCnc2 := RobotIn.Status.bZone_2_CNC_2;
bZoneCnc3 := RobotIn.Status.bZone_3_CNC_3;
bZoneLift1 := RobotIn.Status.bZone_4_Lifter_1;
bZoneLift2 := RobotIn.Status.bZone_5_Lifter_2;
bZoneLift3 := RobotIn.Status.bZone_6_Lifter_3;
bZoneGudel := RobotIn.Status.bZone_7_Gudel;
bZoneMaster := RobotIn.Status.bZone_8_Master;


(*Időzítők***************************************************)
tBaseState(IN:= (nState > 0 AND nState < 10000), PT:= timeBaseState);
tResetFault(IN:= RobotOut.Control.bReset, PT:= T#100MS);
tStopCycle(IN:= RobotOut.Control.bCycleStop, PT:= T#100MS);
tStartCycle(IN:= RobotOut.Control.bStart, PT:= T#100MS);

(*Vész rendszer**************************************************)
bRobotReady :=  NOT RobotIn.Status.bControllerEmyStop AND
				NOT RobotIn.Status.bTeachPendantEmyStop AND
				NOT RobotIn.Status.bDeadman AND
				NOT RobotIn.Status.bFence AND
				NOT RobotIn.Status.bEmyStopExternal;
				
(*Hibakezelés************************************************)
IF nState >= 200 AND nState < 150000 AND (RobotIn.Status.bAlarm OR RobotIn.Status.bFault OR NOT bRobotReady) THEN
	bErrNotReady := TRUE;
ELSIF nState = 40 AND bErrBaseTimeout THEN
	nState := 200000;
END_IF

IF tBaseState.Q AND NOT bErrBaseTimeout THEN
	bErrBaseTimeout := TRUE;
END_IF

bError := (RobotIn.Status.bAlarm AND bEn) OR
			RobotIn.Status.bNoPneumatics OR
			RobotIn.Status.bNotCorrectPrg OR
			RobotIn.Status.bNotProductOnRobot OR
			RobotIn.Status.bProductOnRobot OR
			RobotIn.Status.bGripperOpenError OR
			RobotIn.Status.bGripperCloseError OR
			RobotIn.Status.bOffsetError OR
			RobotIn.Status.bWeightError OR
			bErrNotReady OR
			bErrBaseTimeout;

arrAlarms[0] := RobotIn.Status.bNoPneumatics;			
arrAlarms[1] := RobotIn.Status.bNotCorrectPrg;
arrAlarms[2] := RobotIn.Status.bNotProductOnRobot;
arrAlarms[3] := RobotIn.Status.bProductOnRobot;
arrAlarms[4] := RobotIn.Status.bGripperOpenError;
arrAlarms[5] := RobotIn.Status.bGripperCloseError;
arrAlarms[6] := RobotIn.Status.bOffsetError;
arrAlarms[7] := RobotIn.Status.bWeightError;
arrAlarms[8] := bErrNotReady;
arrAlarms[9] := bErrBaseTimeout;

IF nState > 140 AND nState < 150000 AND bError THEN
	nState := 200000;
END_IF
					
(*State history ************************************************)
IF(nState >= 100) AND (nState <= 20000) THEN
(*Steps before any state*)
	IF anLastStates[0] <> nState THEN
		FOR iLastStates:=500 TO 1 BY -1 DO
			anLastStates[iLastStates]:= anLastStates[iLastStates-1];
		END_FOR
		anLastStates[0]:= nState;
	END_IF
END_IF	

(*Pendant mód ************************************************)
bPendantMode := RobotIn.Status.bPendant;
IF bPendantMode THEN
	nState := 150000;
END_IF

(*Engedélyek *************************************************)
IF (NOT bEn AND NOT bPendantMode) THEN			// nincs ajtókör, és pendantról sem szeretnék használni
	nState := 0;
END_IF

// Enable signals
RobotOut.Control.bZoneEnable := bEn;
RobotOut.Control.bPlcOverride := bOverride;

(*Automata üzem *********************************************)
CASE nState OF
	(* Emergency circuit broken - Base state *)
	0:(* Operation stop - Emergency circuit check *)
		sState := CONCAT(UDINT_TO_STRING(nState) ,' - Vészkör vagy ajtókör bontva - Működtetések törlése');
		RobotOut.Control.bImmediateStop := FALSE;
		RobotOut.Control.bHold := FALSE;
		RobotOut.Control.bSafeSpeed := FALSE;
		RobotOut.Control.bCycleStop := FALSE;
		RobotOut.Control.bReset := FALSE;
		RobotOut.Control.bStart := FALSE;
		RobotOut.Control.bPNS1 := TRUE;
		RobotOut.Control.bPNS2 := FALSE;
		RobotOut.Control.bPNS3 := FALSE;
		RobotOut.Control.bPNS4 := FALSE;
		RobotOut.Control.bPNS5 := FALSE;
		RobotOut.Control.bPNS6 := FALSE;
		RobotOut.Control.bPNS7 := FALSE;
		RobotOut.Control.bPNS8 := FALSE;
		RobotOut.Control.bPnsStrobe := FALSE;
		RobotOut.Control.bEnable := FALSE;
		RobotOut.Control.bHome := FALSE;
		RobotOut.Control.bServiceEnd := FALSE;
		RobotOut.Control.nMode := 0;
		RobotOut.Control.nProgramNumber := 0;
		RobotOut.Control.bProdStart := FALSE;
		RobotOut.Control.bCNC_1_Reset := FALSE;
		RobotOut.Control.bCNC_1_ViseClose_Reset := FALSE;
		RobotOut.Control.bCNC_1_ViseOpen_Reset := FALSE;
		RobotOut.Control.bCNC_2_Reset := FALSE;
		RobotOut.Control.bCNC_2_ViseClose_Reset := FALSE;
		RobotOut.Control.bCNC_2_ViseOpen_Reset := FALSE;
		RobotOut.Control.bCNC_3_Reset := FALSE;
		RobotOut.Control.bCNC_3_ViseClose_Reset := FALSE;
		RobotOut.Control.bCNC_3_ViseOpen_Reset := FALSE;
		RobotOut.Control.bPalette_1_Reset := FALSE;
		RobotOut.Control.bPalette_2_Reset := FALSE;
		RobotOut.Control.bPalette_3_Reset := FALSE;
		RobotOut.Control.bGripperClosed_Reset := FALSE;
		bErrNotReady := FALSE;
		bErrBaseTimeout := FALSE;
		bReady := FALSE;
		bBusy := FALSE;	
		IF bEn AND bRobotReady THEN
			bBusy := TRUE;
			nState := nState + 20;
		END_IF
		
	20:	
		sState := CONCAT(UDINT_TO_STRING(nState) ,' - Alaphelyzetfelvétel - Robot bekapcsolása');
		RobotOut.Control.bImmediateStop := TRUE;
		RobotOut.Control.bHold := TRUE;
		RobotOut.Control.bSafeSpeed := TRUE;
		RobotOut.Control.bEnable := TRUE;
		IF RobotIn.Status.bFault AND NOT RobotOut.Control.bReset THEN
			RobotOut.Control.bReset := TRUE;	// Ha hiba van -> Reset
		END_IF
		nState := nState + 20;

	40:
		sState := CONCAT(UDINT_TO_STRING(nState) ,' - Alaphelyzet felvétel - Robot hibatörlés');	
		IF tResetFault.Q THEN
			RobotOut.Control.bReset := FALSE;
		END_IF
		IF NOT RobotOut.Control.bReset AND NOT RobotIn.Status.bFault THEN
			nState := nState + 20;
		END_IF

	60:
		sState := CONCAT(UDINT_TO_STRING(nState) ,' - Alaphelyzet felvétel - Várakozás Robot hibatörlésre');	
		IF RobotIn.Status.bCommandEnable AND NOT RobotIn.Status.bFault THEN
			nState := nState + 20;
		END_IF
		
	80:
		sState := CONCAT(UDINT_TO_STRING(nState) ,' - Alaphelyzet felvétel - Robot Cycle Stop');
		RobotOut.Control.bCycleStop := TRUE;
		IF tStopCycle.Q THEN
			RobotOut.Control.bCycleStop := FALSE;
			nState := nState + 20;
		END_IF
	
	100:
		sState := CONCAT(UDINT_TO_STRING(nState) ,' - Alaphelyzet felvétel - Robot Cycle Start');
		RobotOut.Control.bStart := TRUE;
		IF tStartCycle.Q THEN
			RobotOut.Control.bStart := FALSE;
			nState := nState + 20;
		END_IF
		
	120: 
		sState := CONCAT(UDINT_TO_STRING(nState) ,' - Alaphelyzet felvétel - Várakozás Robot Cycle Start-ra');
		IF RobotIn.Status.bBusy AND RobotIn.Status.bProgramEnd THEN
			nState := nState + 20;
		END_IF
		
	140:
		sState := CONCAT(UDINT_TO_STRING(nState) ,' - Alaphelyzet felvétel - Alaphelyzet felvétel - Robot Busy');
		IF RobotIn.Status.bBusy THEN
			RobotOut.Control.bProdStart := TRUE;
			nState := nState + 20;
		END_IF
		
	160:
		sState := CONCAT(UDINT_TO_STRING(nState) ,' - Alaphelyzet felvétel - Robot alaphelyzetbe küldése');	
		RobotOut.Control.nProgramNumber := TO_BYTE(E_CNC_Robot_Programs.Home);
		IF RobotOut.Control.nProgramNumber = RobotIn.Status.nProgramNumber THEN
			RobotOut.Control.nProgramNumber := 0;
			nState := nState + 20;
		END_IF
		
	180:
		sState := CONCAT(UDINT_TO_STRING(nState) ,' - Alaphelyzet felvétel - Várakozás a robotprogram végére.');	
		IF RobotIn.Status.bProgramEnd AND NOT RobotIn.Status.bProgramRun THEN
			nState := nState + 20;
		END_IF
		
	200:
		nState := 10000;
		 
(* Alaphelyzet *********************************************************************)
	10000:
		sState := CONCAT(UDINT_TO_STRING(nState) ,' - Alaphelyzet - Várakozás parancsra');
		IF eCommand = E_CNC_Robot_Command.NoCommand THEN
			bReady := TRUE;
			bBusy := FALSE;
			bDone := FALSE;
		ELSE
			bReady := TRUE;
			bBusy := TRUE;
			bDone := FALSE;
			IF eCommand = E_CNC_Robot_Command.Home THEN			
				nState := 11000;	
			ELSIF eCommand = E_CNC_Robot_Command.QuickHome THEN	
				nState := 11500;
			ELSIF eCommand = E_CNC_Robot_Command.Wait THEN	
				nState := 12000;
			ELSIF eCommand = E_CNC_Robot_Command.Service THEN	
				nState := 13000;
			ELSIF eCommand = E_CNC_Robot_Command.Pick_Up_CNC THEN	
				nState := 14000;
			ELSIF eCommand = E_CNC_Robot_Command.Put_Down_CNC THEN	
				nState := 15000;
			ELSIF eCommand = E_CNC_Robot_Command.Pick_Up_Lifter THEN	
				nState := 16000;
			ELSIF eCommand = E_CNC_Robot_Command.Put_Down_Lifter THEN	
				nState := 17000;
			ELSIF eCommand = E_CNC_Robot_Command.Camera_Lifter THEN	
				nState := 18000;
			ELSIF eCommand = E_CNC_Robot_Command.Pick_Up_Master THEN	
				nState := 19000;
			ELSIF eCommand = E_CNC_Robot_Command.Put_Down_Master THEN	
				nState := 20000;
			ELSIF eCommand = E_CNC_Robot_Command.Pick_Up_Master_From_Lifter THEN	
				nState := 21000;
			ELSIF eCommand = E_CNC_Robot_Command.Put_Down_Master_To_Lifter THEN	
				nState := 22000;
			END_IF
		END_IF

{region "Move to Home"} 
	(*-----=== Move to home program végrehajtása ===-----*)
	11000:	
		sState := CONCAT(UDINT_TO_STRING(nState) ,' - Robot alaphelyzetbe küldése');	
		RobotOut.Control.nProgramNumber := TO_BYTE(E_CNC_Robot_Programs.Home);
		IF RobotOut.Control.nProgramNumber = RobotIn.Status.nProgramNumber THEN
			RobotOut.Control.nProgramNumber := 0;
			nState := nState + 20;
		END_IF
		
	11020:
		sState := CONCAT(UDINT_TO_STRING(nState) ,' - Várakozás a robotprogram végére.');	
		IF RobotIn.Status.bProgramEnd AND NOT RobotIn.Status.bProgramRun THEN
			nState := nState + 20;
		END_IF
		
	11040:
		sState := CONCAT(UDINT_TO_STRING(nState) ,' - Várakozás mozgásparancs törlésére.');
		bReady := TRUE;
		bBusy := FALSE;
		bDone := TRUE;
		IF eCommand = E_CNC_Robot_Command.NoCommand THEN
			nState := 10000;
		END_IF
{endregion}

{region "Move to Quick Home"}
	 	(*-----=== Move to quick home program végrehajtása ===-----*)
	11500:	
		sState := CONCAT(UDINT_TO_STRING(nState) ,' - Robot alaphelyzetbe küldése');	
		RobotOut.Control.nProgramNumber := TO_BYTE(E_CNC_Robot_Programs.QuickHome);
		IF RobotOut.Control.nProgramNumber = RobotIn.Status.nProgramNumber THEN
			RobotOut.Control.nProgramNumber := 0;
			nState := nState + 20;
		END_IF
		
	11520:
		sState := CONCAT(UDINT_TO_STRING(nState) ,' - Várakozás a robotprogram végére.');	
		IF RobotIn.Status.bProgramEnd AND NOT RobotIn.Status.bProgramRun THEN
			nState := nState + 20;
		END_IF
		
	11540:
		sState := CONCAT(UDINT_TO_STRING(nState) ,' - Várakozás mozgásparancs törlésére.');
		bReady := TRUE;
		bBusy := FALSE;
		bDone := TRUE;
		IF eCommand = E_CNC_Robot_Command.NoCommand THEN
			nState := 10000;
		END_IF
{endregion}

{region "Move to Wait"}
	(*-----=== Move to wait program végrehajtása ===-----*)
	12000:	
		sState := CONCAT(UDINT_TO_STRING(nState) ,' - Robot várakozó pozícióba küldése');	
		RobotOut.Control.nProgramNumber := TO_BYTE(E_CNC_Robot_Programs.Park);
		IF RobotOut.Control.nProgramNumber = RobotIn.Status.nProgramNumber THEN
			RobotOut.Control.nProgramNumber := 0;
			nState := nState + 20;
		END_IF
		
	12020:
		sState := CONCAT(UDINT_TO_STRING(nState) ,' - Várakozás a robotprogram végére.');	
		IF RobotIn.Status.bProgramEnd AND NOT RobotIn.Status.bProgramRun THEN
			nState := nState + 20;
		END_IF
		
	12040:
		sState := CONCAT(UDINT_TO_STRING(nState) ,' - Várakozás mozgásparancs törlésére.');
		bReady := TRUE;
		bBusy := FALSE;
		bDone := TRUE;
		IF eCommand = E_CNC_Robot_Command.NoCommand THEN
			nState := 10000;
		END_IF
{endregion}
	 
{region "Move to Service"}
	(*-----=== Move to service program végrehajtása ===-----*)
	13000:	
		sState := CONCAT(UDINT_TO_STRING(nState) ,' - Robot szervíz pozícióba küldése');	
		RobotOut.Control.nProgramNumber := TO_BYTE(E_CNC_Robot_Programs.Service);
		IF RobotOut.Control.nProgramNumber = RobotIn.Status.nProgramNumber THEN
			RobotOut.Control.nProgramNumber := 0;
			nState := nState + 20;
		END_IF
		
	13020:
		sState := CONCAT(UDINT_TO_STRING(nState) ,' - Várakozás a robotprogram végére.');	
		IF RobotIn.Status.bProgramEnd AND NOT RobotIn.Status.bProgramRun THEN
			nState := nState + 20;
		END_IF
		
	13040:
		sState := CONCAT(UDINT_TO_STRING(nState) ,' - Várakozás mozgásparancs törlésére.');
		bReady := TRUE;
		bBusy := FALSE;
		bDone := TRUE;
		IF eCommand = E_CNC_Robot_Command.NoCommand THEN
			nState := 10000;
		END_IF
{endregion}
			   
{region "Pick up CNC"}
	(*-----=== CNC pick up program végrehajtása ===-----*)
	14000:	
		sState := CONCAT(UDINT_TO_STRING(nState) ,' - Kivétel CNC-ből');
		REAL_TO_WHOLE_AND_FRACTION(nReal := nOffset_X,
									nWhole => RobotOut.Control.nOffset_X_Whole,
									nFraction => RobotOut.Control.nOffset_X_Fractional);
		REAL_TO_WHOLE_AND_FRACTION(nReal := nOffset_Y,
									nWhole => RobotOut.Control.nOffset_Y_Whole,
									nFraction => RobotOut.Control.nOffset_Y_Fractional);
		REAL_TO_WHOLE_AND_FRACTION(nReal := nOffset_Z,
									nWhole => RobotOut.Control.nOffset_Z_Whole,
									nFraction => RobotOut.Control.nOffset_Z_Fractional);
		REAL_TO_WHOLE_AND_FRACTION(nReal := nOffset_W,
									nWhole => RobotOut.Control.nOffset_W_Whole,
									nFraction => RobotOut.Control.nOffset_W_Fractional);
		REAL_TO_WHOLE_AND_FRACTION(nReal := nOffset_P,
									nWhole => RobotOut.Control.nOffset_P_Whole,
									nFraction => RobotOut.Control.nOffset_P_Fractional);
		REAL_TO_WHOLE_AND_FRACTION(nReal := nOffset_R,
									nWhole => RobotOut.Control.nOffset_R_Whole,
									nFraction => RobotOut.Control.nOffset_R_Fractional);
		IF nCncNumber  = 1 THEN
			RobotOut.Control.nProgramNumber := TO_BYTE(E_CNC_Robot_Programs.CNC_1_PickUp);
		ELSIF nCncNumber  = 2 THEN
			RobotOut.Control.nProgramNumber := TO_BYTE(E_CNC_Robot_Programs.CNC_2_PickUp);
		ELSIF nCncNumber  = 3 THEN
			RobotOut.Control.nProgramNumber := TO_BYTE(E_CNC_Robot_Programs.CNC_3_PickUp);
		END_IF	
		IF RobotOut.Control.nProgramNumber = RobotIn.Status.nProgramNumber THEN
			RobotOut.Control.nProgramNumber := 0;
			nState := nState + 20;
		END_IF
		
	14020:
		sState := CONCAT(UDINT_TO_STRING(nState) ,' - Várakozás a robotprogram végére.');	
		IF RobotIn.Status.bProgramEnd AND NOT RobotIn.Status.bProgramRun THEN
			nState := nState + 20;
		END_IF
		
	14040:
		sState := CONCAT(UDINT_TO_STRING(nState) ,' - Várakozás mozgásparancs törlésére.');
		bReady := TRUE;
		bBusy := FALSE;
		bDone := TRUE;
		IF eCommand = E_CNC_Robot_Command.NoCommand THEN
			nState := 10000;
		END_IF
{endregion}
	 
{region "Put down CNC"}
	(*-----=== CNC put down program végrehajtása ===-----*)
	15000:	
		sState := CONCAT(UDINT_TO_STRING(nState) ,' - Berakás CNC-be');
		REAL_TO_WHOLE_AND_FRACTION(nReal := nOffset_X,
									nWhole => RobotOut.Control.nOffset_X_Whole,
									nFraction => RobotOut.Control.nOffset_X_Fractional);
		REAL_TO_WHOLE_AND_FRACTION(nReal := nOffset_Y,
									nWhole => RobotOut.Control.nOffset_Y_Whole,
									nFraction => RobotOut.Control.nOffset_Y_Fractional);
		REAL_TO_WHOLE_AND_FRACTION(nReal := nOffset_Z,
									nWhole => RobotOut.Control.nOffset_Z_Whole,
									nFraction => RobotOut.Control.nOffset_Z_Fractional);
		REAL_TO_WHOLE_AND_FRACTION(nReal := nOffset_W,
									nWhole => RobotOut.Control.nOffset_W_Whole,
									nFraction => RobotOut.Control.nOffset_W_Fractional);
		REAL_TO_WHOLE_AND_FRACTION(nReal := nOffset_P,
									nWhole => RobotOut.Control.nOffset_P_Whole,
									nFraction => RobotOut.Control.nOffset_P_Fractional);
		REAL_TO_WHOLE_AND_FRACTION(nReal := nOffset_R,
									nWhole => RobotOut.Control.nOffset_R_Whole,
									nFraction => RobotOut.Control.nOffset_R_Fractional);
		IF nCncNumber  = 1 THEN
			RobotOut.Control.nProgramNumber := TO_BYTE(E_CNC_Robot_Programs.CNC_1_PutDown);
		ELSIF nCncNumber  = 2 THEN
			RobotOut.Control.nProgramNumber := TO_BYTE(E_CNC_Robot_Programs.CNC_2_PutDown);
		ELSIF nCncNumber  = 3 THEN
			RobotOut.Control.nProgramNumber := TO_BYTE(E_CNC_Robot_Programs.CNC_3_PutDown);
		END_IF	
		IF RobotOut.Control.nProgramNumber = RobotIn.Status.nProgramNumber THEN
			RobotOut.Control.nProgramNumber := 0;
			nState := nState + 20;
		END_IF
		
	15020:
		sState := CONCAT(UDINT_TO_STRING(nState) ,' - Várakozás a robotprogram végére.');	
		IF RobotIn.Status.bProgramEnd AND NOT RobotIn.Status.bProgramRun THEN
			nState := nState + 20;
		END_IF
		
	15040:
		sState := CONCAT(UDINT_TO_STRING(nState) ,' - Várakozás mozgásparancs törlésére.');
		bReady := TRUE;
		bBusy := FALSE;
		bDone := TRUE;
		IF eCommand = E_CNC_Robot_Command.NoCommand THEN
			nState := 10000;
		END_IF
{endregion}
	 
{region "Pick up Lifter"}
	(*-----=== Lifter pick up program végrehajtása ===-----*)
	16000:	
		sState := CONCAT(UDINT_TO_STRING(nState) ,' - Felvétel kiemelőről');
		REAL_TO_WHOLE_AND_FRACTION(nReal := nOffset_X,
									nWhole => RobotOut.Control.nOffset_X_Whole,
									nFraction => RobotOut.Control.nOffset_X_Fractional);
		REAL_TO_WHOLE_AND_FRACTION(nReal := nOffset_Y,
									nWhole => RobotOut.Control.nOffset_Y_Whole,
									nFraction => RobotOut.Control.nOffset_Y_Fractional);
		REAL_TO_WHOLE_AND_FRACTION(nReal := nOffset_Z,
									nWhole => RobotOut.Control.nOffset_Z_Whole,
									nFraction => RobotOut.Control.nOffset_Z_Fractional);
		REAL_TO_WHOLE_AND_FRACTION(nReal := nOffset_W,
									nWhole => RobotOut.Control.nOffset_W_Whole,
									nFraction => RobotOut.Control.nOffset_W_Fractional);
		REAL_TO_WHOLE_AND_FRACTION(nReal := nOffset_P,
									nWhole => RobotOut.Control.nOffset_P_Whole,
									nFraction => RobotOut.Control.nOffset_P_Fractional);
		REAL_TO_WHOLE_AND_FRACTION(nReal := nOffset_R,
									nWhole => RobotOut.Control.nOffset_R_Whole,
									nFraction => RobotOut.Control.nOffset_R_Fractional);
		IF eLifterNumber  = E_Lifter.Lifter_1A THEN
			RobotOut.Control.nProgramNumber := TO_BYTE(E_CNC_Robot_Programs.Lifter_1A_PickUp);
		ELSIF eLifterNumber  = E_Lifter.Lifter_1B THEN
			RobotOut.Control.nProgramNumber := TO_BYTE(E_CNC_Robot_Programs.Lifter_1B_PickUp);
		ELSIF eLifterNumber  = E_Lifter.Lifter_2A THEN
			RobotOut.Control.nProgramNumber := TO_BYTE(E_CNC_Robot_Programs.Lifter_2A_PickUp);
		ELSIF eLifterNumber  = E_Lifter.Lifter_2B THEN
			RobotOut.Control.nProgramNumber := TO_BYTE(E_CNC_Robot_Programs.Lifter_2B_PickUp);
		ELSIF eLifterNumber  = E_Lifter.Lifter_3A THEN
			RobotOut.Control.nProgramNumber := TO_BYTE(E_CNC_Robot_Programs.Lifter_3A_PickUp);
		ELSIF eLifterNumber  = E_Lifter.Lifter_3B THEN
			RobotOut.Control.nProgramNumber := TO_BYTE(E_CNC_Robot_Programs.Lifter_3B_PickUp);
		END_IF	
		IF RobotOut.Control.nProgramNumber = RobotIn.Status.nProgramNumber THEN
			RobotOut.Control.nProgramNumber := 0;
			nState := nState + 20;
		END_IF
		
	16020:
		sState := CONCAT(UDINT_TO_STRING(nState) ,' - Várakozás a robotprogram végére.');	
		IF RobotIn.Status.bProgramEnd AND NOT RobotIn.Status.bProgramRun THEN
			nState := nState + 20;
		END_IF
		
	16040:
		sState := CONCAT(UDINT_TO_STRING(nState) ,' - Várakozás mozgásparancs törlésére.');
		bReady := TRUE;
		bBusy := FALSE;
		bDone := TRUE;
		IF eCommand = E_CNC_Robot_Command.NoCommand THEN
			nState := 10000;
		END_IF
{endregion}
	 
{region "Put down Lifter"}
	(*-----=== Lifter put down program végrehajtása ===-----*)
	17000:	
		sState := CONCAT(UDINT_TO_STRING(nState) ,' - Lerakás kiemelőre');
		IF eLifterNumber  = E_Lifter.Lifter_1A THEN
			RobotOut.Control.nProgramNumber := TO_BYTE(E_CNC_Robot_Programs.Lifter_1A_PutDown);
		ELSIF eLifterNumber  = E_Lifter.Lifter_1B THEN
			RobotOut.Control.nProgramNumber := TO_BYTE(E_CNC_Robot_Programs.Lifter_1B_PutDown);
		ELSIF eLifterNumber  = E_Lifter.Lifter_2A THEN
			RobotOut.Control.nProgramNumber := TO_BYTE(E_CNC_Robot_Programs.Lifter_2A_PutDown);
		ELSIF eLifterNumber  = E_Lifter.Lifter_2B THEN
			RobotOut.Control.nProgramNumber := TO_BYTE(E_CNC_Robot_Programs.Lifter_2B_PutDown);
		ELSIF eLifterNumber  = E_Lifter.Lifter_3A THEN
			RobotOut.Control.nProgramNumber := TO_BYTE(E_CNC_Robot_Programs.Lifter_3A_PutDown);
		ELSIF eLifterNumber  = E_Lifter.Lifter_3B THEN
			RobotOut.Control.nProgramNumber := TO_BYTE(E_CNC_Robot_Programs.Lifter_3B_PutDown);
		END_IF	
		IF RobotOut.Control.nProgramNumber = RobotIn.Status.nProgramNumber THEN
			RobotOut.Control.nProgramNumber := 0;
			nState := nState + 20;
		END_IF
		
	17020:
		sState := CONCAT(UDINT_TO_STRING(nState) ,' - Várakozás a robotprogram végére.');	
		IF RobotIn.Status.bProgramEnd AND NOT RobotIn.Status.bProgramRun THEN
			nState := nState + 20;
		END_IF
		
	17040:
		sState := CONCAT(UDINT_TO_STRING(nState) ,' - Várakozás mozgásparancs törlésére.');
		bReady := TRUE;
		bBusy := FALSE;
		bDone := TRUE;
		IF eCommand = E_CNC_Robot_Command.NoCommand THEN
			nState := 10000;
		END_IF
{endregion}
	 
{region "Camera Lifter"}
	(*-----=== Lifter camera program végrehajtása ===-----*)
	18000:	
		sState := CONCAT(UDINT_TO_STRING(nState) ,' - Kamerázás kiemelőnél');
		IF eLifterNumber  = E_Lifter.Lifter_1A THEN
			RobotOut.Control.nProgramNumber := TO_BYTE(E_CNC_Robot_Programs.Lifter_1A_Camera);
		ELSIF eLifterNumber  = E_Lifter.Lifter_1B THEN
			RobotOut.Control.nProgramNumber := TO_BYTE(E_CNC_Robot_Programs.Lifter_1B_Camera);
		ELSIF eLifterNumber  = E_Lifter.Lifter_2A THEN
			RobotOut.Control.nProgramNumber := TO_BYTE(E_CNC_Robot_Programs.Lifter_2A_Camera);
		ELSIF eLifterNumber  = E_Lifter.Lifter_2B THEN
			RobotOut.Control.nProgramNumber := TO_BYTE(E_CNC_Robot_Programs.Lifter_2B_Camera);
		ELSIF eLifterNumber  = E_Lifter.Lifter_3A THEN
			RobotOut.Control.nProgramNumber := TO_BYTE(E_CNC_Robot_Programs.Lifter_3A_Camera);
		ELSIF eLifterNumber  = E_Lifter.Lifter_3B THEN
			RobotOut.Control.nProgramNumber := TO_BYTE(E_CNC_Robot_Programs.Lifter_3B_Camera);
		END_IF
		IF RobotOut.Control.nProgramNumber = RobotIn.Status.nProgramNumber THEN
			RobotOut.Control.nProgramNumber := 0;
			nState := nState + 20;
		END_IF
		
	18020:
		sState := CONCAT(UDINT_TO_STRING(nState) ,' - Várakozás a robotprogram végére.');	
		IF RobotIn.Status.bProgramEnd AND NOT RobotIn.Status.bProgramRun THEN
			nState := nState + 20;
		END_IF
		
	18040:
		sState := CONCAT(UDINT_TO_STRING(nState) ,' - Várakozás mozgásparancs törlésére.');
		bReady := TRUE;
		bBusy := FALSE;
		bDone := TRUE;
		IF eCommand = E_CNC_Robot_Command.NoCommand THEN
			nState := 10000;
		END_IF
{endregion}
								   
{region "Pick up Master"}
	(*-----=== Master pick up program végrehajtása ===-----*)
	19000:	
		sState := CONCAT(UDINT_TO_STRING(nState) ,' - Mester darab felvétele');
		RobotOut.Control.nOffset_ID := nOffset_ID;
		REAL_TO_WHOLE_AND_FRACTION(nReal := nOffset_X,
									nWhole => RobotOut.Control.nOffset_X_Whole,
									nFraction => RobotOut.Control.nOffset_X_Fractional);
		REAL_TO_WHOLE_AND_FRACTION(nReal := nOffset_Y,
									nWhole => RobotOut.Control.nOffset_Y_Whole,
									nFraction => RobotOut.Control.nOffset_Y_Fractional);
		REAL_TO_WHOLE_AND_FRACTION(nReal := nOffset_Z,
									nWhole => RobotOut.Control.nOffset_Z_Whole,
									nFraction => RobotOut.Control.nOffset_Z_Fractional);
		REAL_TO_WHOLE_AND_FRACTION(nReal := nOffset_W,
									nWhole => RobotOut.Control.nOffset_W_Whole,
									nFraction => RobotOut.Control.nOffset_W_Fractional);
		REAL_TO_WHOLE_AND_FRACTION(nReal := nOffset_P,
									nWhole => RobotOut.Control.nOffset_P_Whole,
									nFraction => RobotOut.Control.nOffset_P_Fractional);
		REAL_TO_WHOLE_AND_FRACTION(nReal := nOffset_R,
									nWhole => RobotOut.Control.nOffset_R_Whole,
									nFraction => RobotOut.Control.nOffset_R_Fractional);
		RobotOut.Control.nProgramNumber := TO_BYTE(E_CNC_Robot_Programs.Master_Part_PickUp);
		IF RobotOut.Control.nProgramNumber = RobotIn.Status.nProgramNumber THEN
			RobotOut.Control.nProgramNumber := 0;
			nState := nState + 20;
		END_IF
		
	19020:
		sState := CONCAT(UDINT_TO_STRING(nState) ,' - Várakozás a robotprogram végére.');	
		IF RobotIn.Status.bProgramEnd AND NOT RobotIn.Status.bProgramRun THEN
			nState := nState + 20;
		END_IF
		
	19040:
		sState := CONCAT(UDINT_TO_STRING(nState) ,' - Várakozás mozgásparancs törlésére.');
		bReady := TRUE;
		bBusy := FALSE;
		bDone := TRUE;
		IF eCommand = E_CNC_Robot_Command.NoCommand THEN
			nState := 10000;
		END_IF
{endregion}
	 
{region "Put down Master"}
	(*-----=== Master put down program végrehajtása ===-----*)
	20000:	
		sState := CONCAT(UDINT_TO_STRING(nState) ,' - Mester darab lerakása');
		REAL_TO_WHOLE_AND_FRACTION(nReal := nOffset_X,
									nWhole => RobotOut.Control.nOffset_X_Whole,
									nFraction => RobotOut.Control.nOffset_X_Fractional);
		REAL_TO_WHOLE_AND_FRACTION(nReal := nOffset_Y,
									nWhole => RobotOut.Control.nOffset_Y_Whole,
									nFraction => RobotOut.Control.nOffset_Y_Fractional);
		REAL_TO_WHOLE_AND_FRACTION(nReal := nOffset_Z,
									nWhole => RobotOut.Control.nOffset_Z_Whole,
									nFraction => RobotOut.Control.nOffset_Z_Fractional);
		REAL_TO_WHOLE_AND_FRACTION(nReal := nOffset_W,
									nWhole => RobotOut.Control.nOffset_W_Whole,
									nFraction => RobotOut.Control.nOffset_W_Fractional);
		REAL_TO_WHOLE_AND_FRACTION(nReal := nOffset_P,
									nWhole => RobotOut.Control.nOffset_P_Whole,
									nFraction => RobotOut.Control.nOffset_P_Fractional);
		REAL_TO_WHOLE_AND_FRACTION(nReal := nOffset_R,
									nWhole => RobotOut.Control.nOffset_R_Whole,
									nFraction => RobotOut.Control.nOffset_R_Fractional);
		RobotOut.Control.nProgramNumber := TO_BYTE(E_CNC_Robot_Programs.Master_Part_PutDown);
		IF RobotOut.Control.nProgramNumber = RobotIn.Status.nProgramNumber THEN
			RobotOut.Control.nProgramNumber := 0;
			nState := nState + 20;
		END_IF
		
	20020:
		sState := CONCAT(UDINT_TO_STRING(nState) ,' - Várakozás a robotprogram végére.');	
		IF RobotIn.Status.bProgramEnd AND NOT RobotIn.Status.bProgramRun THEN
			nState := nState + 20;
		END_IF
		
	20040:
		sState := CONCAT(UDINT_TO_STRING(nState) ,' - Várakozás mozgásparancs törlésére.');
		bReady := TRUE;
		bBusy := FALSE;
		bDone := TRUE;
		IF eCommand = E_CNC_Robot_Command.NoCommand THEN
			nState := 10000;
		END_IF
{endregion}
											 
{region "Pick up Master from Lifter"}
	(*-----=== Pick up Master from Lifter program végrehajtása ===-----*)
	21000:	
		sState := CONCAT(UDINT_TO_STRING(nState) ,' - Mester felvétel kiemelőből');
		REAL_TO_WHOLE_AND_FRACTION(nReal := nOffset_X,
									nWhole => RobotOut.Control.nOffset_X_Whole,
									nFraction => RobotOut.Control.nOffset_X_Fractional);
		REAL_TO_WHOLE_AND_FRACTION(nReal := nOffset_Y,
									nWhole => RobotOut.Control.nOffset_Y_Whole,
									nFraction => RobotOut.Control.nOffset_Y_Fractional);
		REAL_TO_WHOLE_AND_FRACTION(nReal := nOffset_Z,
									nWhole => RobotOut.Control.nOffset_Z_Whole,
									nFraction => RobotOut.Control.nOffset_Z_Fractional);
		REAL_TO_WHOLE_AND_FRACTION(nReal := nOffset_W,
									nWhole => RobotOut.Control.nOffset_W_Whole,
									nFraction => RobotOut.Control.nOffset_W_Fractional);
		REAL_TO_WHOLE_AND_FRACTION(nReal := nOffset_P,
									nWhole => RobotOut.Control.nOffset_P_Whole,
									nFraction => RobotOut.Control.nOffset_P_Fractional);
		REAL_TO_WHOLE_AND_FRACTION(nReal := nOffset_R,
									nWhole => RobotOut.Control.nOffset_R_Whole,
									nFraction => RobotOut.Control.nOffset_R_Fractional);													   
		IF eLifterNumber  = E_Lifter.Lifter_1A THEN
			RobotOut.Control.nProgramNumber := TO_BYTE(E_CNC_Robot_Programs.Lifter_1A_Master_PickUp);
		ELSIF eLifterNumber  = E_Lifter.Lifter_1B THEN
			RobotOut.Control.nProgramNumber := TO_BYTE(E_CNC_Robot_Programs.Lifter_1B_Master_PickUp);
		ELSIF eLifterNumber  = E_Lifter.Lifter_2A THEN
			RobotOut.Control.nProgramNumber := TO_BYTE(E_CNC_Robot_Programs.Lifter_2A_Master_PickUp);
		ELSIF eLifterNumber  = E_Lifter.Lifter_2B THEN
			RobotOut.Control.nProgramNumber := TO_BYTE(E_CNC_Robot_Programs.Lifter_2B_Master_PickUp);
		ELSIF eLifterNumber  = E_Lifter.Lifter_3A THEN
			RobotOut.Control.nProgramNumber := TO_BYTE(E_CNC_Robot_Programs.Lifter_3A_Master_PickUp);
		ELSIF eLifterNumber  = E_Lifter.Lifter_3B THEN
			RobotOut.Control.nProgramNumber := TO_BYTE(E_CNC_Robot_Programs.Lifter_3B_Master_PickUp);
		END_IF
		IF RobotOut.Control.nProgramNumber = RobotIn.Status.nProgramNumber THEN
			RobotOut.Control.nProgramNumber := 0;
			nState := nState + 20;
		END_IF
		
	21020:
		sState := CONCAT(UDINT_TO_STRING(nState) ,' - Várakozás a robotprogram végére.');	
		IF RobotIn.Status.bProgramEnd AND NOT RobotIn.Status.bProgramRun THEN
			nState := nState + 20;
		END_IF
		
	21040:
		sState := CONCAT(UDINT_TO_STRING(nState) ,' - Várakozás mozgásparancs törlésére.');
		bReady := TRUE;
		bBusy := FALSE;
		bDone := TRUE;
		IF eCommand = E_CNC_Robot_Command.NoCommand THEN
			nState := 10000;
		END_IF
{endregion}
	 
{region "Put down Master to Lifter"}
	(*-----=== Put down Master to Lifter program végrehajtása ===-----*)
	22000:	
		sState := CONCAT(UDINT_TO_STRING(nState) ,' - Mester lerakás kiemelőbe');
		REAL_TO_WHOLE_AND_FRACTION(nReal := nOffset_X,
									nWhole => RobotOut.Control.nOffset_X_Whole,
									nFraction => RobotOut.Control.nOffset_X_Fractional);
		REAL_TO_WHOLE_AND_FRACTION(nReal := nOffset_Y,
									nWhole => RobotOut.Control.nOffset_Y_Whole,
									nFraction => RobotOut.Control.nOffset_Y_Fractional);
		REAL_TO_WHOLE_AND_FRACTION(nReal := nOffset_Z,
									nWhole => RobotOut.Control.nOffset_Z_Whole,
									nFraction => RobotOut.Control.nOffset_Z_Fractional);
		REAL_TO_WHOLE_AND_FRACTION(nReal := nOffset_W,
									nWhole => RobotOut.Control.nOffset_W_Whole,
									nFraction => RobotOut.Control.nOffset_W_Fractional);
		REAL_TO_WHOLE_AND_FRACTION(nReal := nOffset_P,
									nWhole => RobotOut.Control.nOffset_P_Whole,
									nFraction => RobotOut.Control.nOffset_P_Fractional);
		REAL_TO_WHOLE_AND_FRACTION(nReal := nOffset_R,
									nWhole => RobotOut.Control.nOffset_R_Whole,
									nFraction => RobotOut.Control.nOffset_R_Fractional);
		IF eLifterNumber  = E_Lifter.Lifter_1A THEN
			RobotOut.Control.nProgramNumber := TO_BYTE(E_CNC_Robot_Programs.Lifter_1A_Master_PutDown);
		ELSIF eLifterNumber  = E_Lifter.Lifter_1B THEN
			RobotOut.Control.nProgramNumber := TO_BYTE(E_CNC_Robot_Programs.Lifter_1B_Master_PutDown);
		ELSIF eLifterNumber  = E_Lifter.Lifter_2A THEN
			RobotOut.Control.nProgramNumber := TO_BYTE(E_CNC_Robot_Programs.Lifter_2A_Master_PutDown);
		ELSIF eLifterNumber  = E_Lifter.Lifter_2B THEN
			RobotOut.Control.nProgramNumber := TO_BYTE(E_CNC_Robot_Programs.Lifter_2B_Master_PutDown);
		ELSIF eLifterNumber  = E_Lifter.Lifter_3A THEN
			RobotOut.Control.nProgramNumber := TO_BYTE(E_CNC_Robot_Programs.Lifter_3A_Master_PutDown);
		ELSIF eLifterNumber  = E_Lifter.Lifter_3B THEN
			RobotOut.Control.nProgramNumber := TO_BYTE(E_CNC_Robot_Programs.Lifter_3B_Master_PutDown);
		END_IF
		IF RobotOut.Control.nProgramNumber = RobotIn.Status.nProgramNumber THEN
			RobotOut.Control.nProgramNumber := 0;
			nState := nState + 20;
		END_IF
		
	22020:
		sState := CONCAT(UDINT_TO_STRING(nState) ,' - Várakozás a robotprogram végére.');	
		IF RobotIn.Status.bProgramEnd AND NOT RobotIn.Status.bProgramRun THEN
			nState := nState + 20;
		END_IF
		
	22040:
		sState := CONCAT(UDINT_TO_STRING(nState) ,' - Várakozás mozgásparancs törlésére.');
		bReady := TRUE;
		bBusy := FALSE;
		bDone := TRUE;
		IF eCommand = E_CNC_Robot_Command.NoCommand THEN
			nState := 10000;
		END_IF
{endregion}
	 
{region "Pendant mode"}
(* Pendant mód *********************************************************************)
	150000:	sState := CONCAT(UDINT_TO_STRING(nState) ,' - Pendant mód');
			IF NOT bPendantMode THEN
				RobotOut.Control.bImmediateStop := FALSE;
				RobotOut.Control.bHold := FALSE;
				RobotOut.Control.bZoneEnable := FALSE;
				RobotOut.Control.bEnable := FALSE;
				nState := 0;
			ELSE
				RobotOut.Control.bEnable := TRUE;
				RobotOut.Control.bHold := TRUE;
				RobotOut.Control.bZoneEnable := TRUE;
				RobotOut.Control.bImmediateStop := TRUE;
			END_IF
{endregion}
		
(* Hibakezelés *********************************************************************)
	200000:	sState := CONCAT(UDINT_TO_STRING(nState) ,CONCAT(' - Hiba, ebből az állapotból: ' ,sState));
			bReady := FALSE;
			bBusy := FALSE;	
			nState := nState + 20;

(* Hibakezelés *********************************************************************)
	200020:	
			IF bAck THEN			
				nState := nState + 20;
			END_IF
			
	200040: 
			RobotOut.Control.bImmediateStop := TRUE;
			RobotOut.Control.bReset := TRUE;
			RobotOut.Control.bNotCorrectPrg_Reset := TRUE;
			RobotOut.Control.bNotProductOnRobot_Reset := TRUE;
			RobotOut.Control.bProductOnRobot_Reset := TRUE;
			RobotOut.Control.bGripperOpenError_Reset := TRUE;
			RobotOut.Control.bGripperCloseError_Reset := TRUE;
			RobotOut.Control.bOffsetError_Reset := TRUE;
			RobotOut.Control.bWeightError_Reset := TRUE;
			nState := nState + 20;
			
	200060:
			IF 	NOT RobotIn.Status.bNoPneumatics AND
				NOT RobotIn.Status.bNotCorrectPrg AND
				NOT RobotIn.Status.bNotProductOnRobot AND
				NOT RobotIn.Status.bProductOnRobot AND
				NOT RobotIn.Status.bGripperOpenError AND
				NOT RobotIn.Status.bGripperCloseError AND
				NOT RobotIn.Status.bOffsetError AND
				NOT	RobotIn.Status.bWeightError													 
			THEN
				nState := nState + 20;
			END_IF	
			
	200080:
			RobotOut.Control.bReset := FALSE;
			RobotOut.Control.bNotCorrectPrg_Reset := FALSE;
			RobotOut.Control.bNotProductOnRobot_Reset := FALSE;
			RobotOut.Control.bProductOnRobot_Reset := FALSE;
			RobotOut.Control.bGripperOpenError_Reset := FALSE;
			RobotOut.Control.bGripperCloseError_Reset := FALSE;
			RobotOut.Control.bOffsetError_Reset := FALSE;
			RobotOut.Control.bWeightError_Reset := FALSE;
			bErrNotReady := FALSE;
			bErrBaseTimeout := FALSE;
			nState := 0;
ELSE
	sState := CONCAT(UDINT_TO_STRING(nState) ,' - Nem használt állapot');
END_CASE	


(*Hiba string*)
IF bError THEN
	sError := sName;
	FOR i:=0 TO nMaxAlarmNr DO
		IF arrAlarms[i] THEN
			IF (fbAlarmArray[i].eConfirmationState <> 2 AND fbAlarmArray[i].nTimeCleared <> 0 AND fbAlarmArray[i].nTimeConfirmed <> 0) OR //Ha már volt alarm, akkor van bennük érték
				(fbAlarmArray[i].eConfirmationState = 1 AND fbAlarmArray[i].nTimeCleared = 0 AND fbAlarmArray[i].nTimeConfirmed = 0)	//Első futás esetén
			THEN
				fbAlarmArray[i].Raise(0);
			END_IF
		END_IF
	END_FOR 
ELSE
	sError := '';
END_IF

(*Hiba kezelés Tc3_EventLogger*)
IF NOT bIsInitalized THEN
	bIsInitalized := TRUE;
	FOR i:=0 TO nMaxAlarmNr DO
		fbAlarmArray[i].CreateEx(stEventArray[i], TRUE, 0);
	END_FOR
END_IF

(*Hiba törlés (nyugtázott és megszűnt)*)
FOR i:=0 TO nMaxAlarmNr DO
	IF fbAlarmArray[i].eConfirmationState = 3 AND NOT bError THEN
		fbAlarmArray[i].Clear(0, FALSE);
	END_IF
END_FOR

